LIN {X 33.675,Y 43.444,Z 52.000,A 180.000,B 0.000,C 180.000} C_DIS
LIN {X 33.433,Y 43.340,Z 52.000,A 180.000,B 0.000,C 180.000} C_DIS
LIN {X 33.269,Y 43.266,Z 52.000,A 180.000,B 0.000,C 180.000} C_DIS
LIN {X 32.897,Y 43.076,Z 52.000,A 180.000,B 0.000,C 180.000} C_DIS
LIN {X 32.718,Y 42.971,Z 52.000,A 180.000,B 0.000,C 180.000} C_DIS
LIN {X 32.539,Y 42.865,Z 52.000,A 180.000,B 0.000,C 180.000} C_DIS
LIN {X 32.361,Y 42.749,Z 52.000,A 180.000,B 0.000,C 180.000} C_DIS
LIN {X 32.182,Y 42.627,Z 52.000,A 180.000,B 0.000,C 180.000} C_DIS
LIN {X 32.072,Y 42.550,Z 52.000,A 180.000,B 0.000,C 180.000} C_DIS
LIN {X 31.824,Y 42.359,Z 52.000,A 180.000,B 0.000,C 180.000} C_DIS
LIN {X 31.646,Y 42.212,Z 52.000,A 180.000,B 0.000,C 180.000} C_DIS
LIN {X 31.421,Y 42.014,Z 52.000,A 180.000,B 0.000,C 180.000} C_DIS
LIN {X 31.288,Y 41.888,Z 52.000,A 180.000,B 0.000,C 180.000} C_DIS
LIN {X 31.057,Y 41.657,Z 52.000,A 180.000,B 0.000,C 180.000} C_DIS
LIN {X 30.930,Y 41.516,Z 52.000,A 180.000,B 0.000,C 180.000} C_DIS
LIN {X 30.739,Y 41.299,Z 52.000,A 180.000,B 0.000,C 180.000} C_DIS
LIN {X 30.598,Y 41.120,Z 52.000,A 180.000,B 0.000,C 180.000} C_DIS
LIN {X 30.460,Y 40.942,Z 52.000,A 180.000,B 0.000,C 180.000} C_DIS
LIN {X 30.394,Y 40.850,Z 52.000,A 180.000,B 0.000,C 180.000} C_DIS
LIN {X 30.213,Y 40.584,Z 52.000,A 180.000,B 0.000,C 180.000} C_DIS
LIN {X 30.102,Y 40.405,Z 52.000,A 180.000,B 0.000,C 180.000} C_DIS
LIN {X 29.996,Y 40.226,Z 52.000,A 180.000,B 0.000,C 180.000} C_DIS
LIN {X 29.896,Y 40.048,Z 52.000,A 180.000,B 0.000,C 180.000} C_DIS
LIN {X 29.805,Y 39.869,Z 52.000,A 180.000,B 0.000,C 180.000} C_DIS
LIN {X 29.714,Y 39.690,Z 52.000,A 180.000,B 0.000,C 180.000} C_DIS
LIN {X 29.559,Y 39.333,Z 52.000,A 180.000,B 0.000,C 180.000} C_DIS
LIN {X 29.500,Y 39.184,Z 52.000,A 180.000,B 0.000,C 180.000} C_DIS
LIN {X 29.425,Y 38.975,Z 52.000,A 180.000,B 0.000,C 180.000} C_DIS
LIN {X 29.362,Y 38.796,Z 52.000,A 180.000,B 0.000,C 180.000} C_DIS
LIN {X 29.258,Y 38.439,Z 52.000,A 180.000,B 0.000,C 180.000} C_DIS
LIN {X 29.213,Y 38.260,Z 52.000,A 180.000,B 0.000,C 180.000} C_DIS
LIN {X 29.143,Y 37.944,Z 52.000,A 180.000,B 0.000,C 180.000} C_DIS
LIN {X 29.134,Y 37.902,Z 52.000,A 180.000,B 0.000,C 180.000} C_DIS
LIN {X 29.077,Y 37.545,Z 52.000,A 180.000,B 0.000,C 180.000} C_DIS
LIN {X 29.053,Y 37.366,Z 52.000,A 180.000,B 0.000,C 180.000} C_DIS
LIN {X 29.020,Y 37.009,Z 52.000,A 180.000,B 0.000,C 180.000} C_DIS
LIN {X 29.012,Y 36.830,Z 52.000,A 180.000,B 0.000,C 180.000} C_DIS
LIN {X 29.006,Y 36.651,Z 52.000,A 180.000,B 0.000,C 180.000} C_DIS
LIN {X 29.002,Y 36.472,Z 52.000,A 180.000,B 0.000,C 180.000} C_DIS
LIN {X 29.013,Y 36.115,Z 52.000,A 180.000,B 0.000,C 180.000} C_DIS
LIN {X 29.025,Y 35.936,Z 52.000,A 180.000,B 0.000,C 180.000} C_DIS
LIN {X 29.059,Y 35.578,Z 52.000,A 180.000,B 0.000,C 180.000} C_DIS
LIN {X 29.086,Y 35.400,Z 52.000,A 180.000,B 0.000,C 180.000} C_DIS
LIN {X 29.114,Y 35.221,Z 52.000,A 180.000,B 0.000,C 180.000} C_DIS
LIN {X 29.143,Y 35.056,Z 52.000,A 180.000,B 0.000,C 180.000} C_DIS
LIN {X 29.226,Y 34.685,Z 52.000,A 180.000,B 0.000,C 180.000} C_DIS
LIN {X 29.274,Y 34.506,Z 52.000,A 180.000,B 0.000,C 180.000} C_DIS
LIN {X 29.326,Y 34.327,Z 52.000,A 180.000,B 0.000,C 180.000} C_DIS
LIN {X 29.381,Y 34.148,Z 52.000,A 180.000,B 0.000,C 180.000} C_DIS
LIN {X 29.509,Y 33.791,Z 52.000,A 180.000,B 0.000,C 180.000} C_DIS
LIN {X 29.583,Y 33.612,Z 52.000,A 180.000,B 0.000,C 180.000} C_DIS
LIN {X 29.679,Y 33.390,Z 52.000,A 180.000,B 0.000,C 180.000} C_DIS
LIN {X 29.742,Y 33.254,Z 52.000,A 180.000,B 0.000,C 180.000} C_DIS
LIN {X 29.924,Y 32.897,Z 52.000,A 180.000,B 0.000,C 180.000} C_DIS
LIN {X 30.029,Y 32.718,Z 52.000,A 180.000,B 0.000,C 180.000} C_DIS
LIN {X 30.135,Y 32.539,Z 52.000,A 180.000,B 0.000,C 180.000} C_DIS
LIN {X 30.215,Y 32.413,Z 52.000,A 180.000,B 0.000,C 180.000} C_DIS
LIN {X 30.394,Y 32.150,Z 52.000,A 180.000,B 0.000,C 180.000} C_DIS
LIN {X 30.503,Y 32.003,Z 52.000,A 180.000,B 0.000,C 180.000} C_DIS
LIN {X 30.641,Y 31.824,Z 52.000,A 180.000,B 0.000,C 180.000} C_DIS
LIN {X 30.752,Y 31.687,Z 52.000,A 180.000,B 0.000,C 180.000} C_DIS
LIN {X 30.945,Y 31.467,Z 52.000,A 180.000,B 0.000,C 180.000} C_DIS
LIN {X 31.109,Y 31.291,Z 52.000,A 180.000,B 0.000,C 180.000} C_DIS
LIN {X 31.291,Y 31.109,Z 52.000,A 180.000,B 0.000,C 180.000} C_DIS
LIN {X 31.467,Y 30.945,Z 52.000,A 180.000,B 0.000,C 180.000} C_DIS
LIN {X 31.687,Y 30.752,Z 52.000,A 180.000,B 0.000,C 180.000} C_DIS
LIN {X 31.824,Y 30.641,Z 52.000,A 180.000,B 0.000,C 180.000} C_DIS
LIN {X 32.003,Y 30.503,Z 52.000,A 180.000,B 0.000,C 180.000} C_DIS
LIN {X 32.150,Y 30.394,Z 52.000,A 180.000,B 0.000,C 180.000} C_DIS
LIN {X 32.413,Y 30.215,Z 52.000,A 180.000,B 0.000,C 180.000} C_DIS
LIN {X 32.539,Y 30.135,Z 52.000,A 180.000,B 0.000,C 180.000} C_DIS
LIN {X 32.718,Y 30.029,Z 52.000,A 180.000,B 0.000,C 180.000} C_DIS
LIN {X 32.897,Y 29.924,Z 52.000,A 180.000,B 0.000,C 180.000} C_DIS
LIN {X 33.254,Y 29.742,Z 52.000,A 180.000,B 0.000,C 180.000} C_DIS
LIN {X 33.390,Y 29.679,Z 52.000,A 180.000,B 0.000,C 180.000} C_DIS
LIN {X 33.612,Y 29.583,Z 52.000,A 180.000,B 0.000,C 180.000} C_DIS
LIN {X 33.791,Y 29.509,Z 52.000,A 180.000,B 0.000,C 180.000} C_DIS
LIN {X 34.148,Y 29.381,Z 52.000,A 180.000,B 0.000,C 180.000} C_DIS
LIN {X 34.327,Y 29.326,Z 52.000,A 180.000,B 0.000,C 180.000} C_DIS
LIN {X 34.506,Y 29.274,Z 52.000,A 180.000,B 0.000,C 180.000} C_DIS
LIN {X 34.685,Y 29.226,Z 52.000,A 180.000,B 0.000,C 180.000} C_DIS
LIN {X 35.056,Y 29.143,Z 52.000,A 180.000,B 0.000,C 180.000} C_DIS
LIN {X 35.221,Y 29.114,Z 52.000,A 180.000,B 0.000,C 180.000} C_DIS
LIN {X 35.400,Y 29.086,Z 52.000,A 180.000,B 0.000,C 180.000} C_DIS
LIN {X 35.578,Y 29.059,Z 52.000,A 180.000,B 0.000,C 180.000} C_DIS
LIN {X 35.936,Y 29.025,Z 52.000,A 180.000,B 0.000,C 180.000} C_DIS
LIN {X 36.115,Y 29.013,Z 52.000,A 180.000,B 0.000,C 180.000} C_DIS
LIN {X 36.472,Y 29.002,Z 52.000,A 180.000,B 0.000,C 180.000} C_DIS
LIN {X 36.651,Y 29.006,Z 52.000,A 180.000,B 0.000,C 180.000} C_DIS
LIN {X 36.830,Y 29.012,Z 52.000,A 180.000,B 0.000,C 180.000} C_DIS
LIN {X 37.009,Y 29.020,Z 52.000,A 180.000,B 0.000,C 180.000} C_DIS
LIN {X 37.366,Y 29.053,Z 52.000,A 180.000,B 0.000,C 180.000} C_DIS
LIN {X 37.545,Y 29.077,Z 52.000,A 180.000,B 0.000,C 180.000} C_DIS
LIN {X 37.902,Y 29.134,Z 52.000,A 180.000,B 0.000,C 180.000} C_DIS
LIN {X 37.944,Y 29.143,Z 52.000,A 180.000,B 0.000,C 180.000} C_DIS
LIN {X 38.260,Y 29.213,Z 52.000,A 180.000,B 0.000,C 180.000} C_DIS
LIN {X 38.439,Y 29.258,Z 52.000,A 180.000,B 0.000,C 180.000} C_DIS
LIN {X 38.796,Y 29.362,Z 52.000,A 180.000,B 0.000,C 180.000} C_DIS
LIN {X 38.975,Y 29.425,Z 52.000,A 180.000,B 0.000,C 180.000} C_DIS
LIN {X 39.184,Y 29.500,Z 52.000,A 180.000,B 0.000,C 180.000} C_DIS
LIN {X 39.333,Y 29.559,Z 52.000,A 180.000,B 0.000,C 180.000} C_DIS
LIN {X 39.690,Y 29.714,Z 52.000,A 180.000,B 0.000,C 180.000} C_DIS
LIN {X 39.869,Y 29.805,Z 52.000,A 180.000,B 0.000,C 180.000} C_DIS
LIN {X 40.048,Y 29.896,Z 52.000,A 180.000,B 0.000,C 180.000} C_DIS
LIN {X 40.226,Y 29.996,Z 52.000,A 180.000,B 0.000,C 180.000} C_DIS
LIN {X 40.405,Y 30.102,Z 52.000,A 180.000,B 0.000,C 180.000} C_DIS
LIN {X 40.584,Y 30.213,Z 52.000,A 180.000,B 0.000,C 180.000} C_DIS
LIN {X 40.850,Y 30.394,Z 52.000,A 180.000,B 0.000,C 180.000} C_DIS
LIN {X 40.942,Y 30.460,Z 52.000,A 180.000,B 0.000,C 180.000} C_DIS
LIN {X 41.120,Y 30.598,Z 52.000,A 180.000,B 0.000,C 180.000} C_DIS
LIN {X 41.299,Y 30.739,Z 52.000,A 180.000,B 0.000,C 180.000} C_DIS
LIN {X 41.516,Y 30.930,Z 52.000,A 180.000,B 0.000,C 180.000} C_DIS
LIN {X 41.657,Y 31.057,Z 52.000,A 180.000,B 0.000,C 180.000} C_DIS
LIN {X 41.888,Y 31.288,Z 52.000,A 180.000,B 0.000,C 180.000} C_DIS
LIN {X 42.014,Y 31.421,Z 52.000,A 180.000,B 0.000,C 180.000} C_DIS
LIN {X 42.212,Y 31.646,Z 52.000,A 180.000,B 0.000,C 180.000} C_DIS
LIN {X 42.359,Y 31.824,Z 52.000,A 180.000,B 0.000,C 180.000} C_DIS
LIN {X 42.550,Y 32.072,Z 52.000,A 180.000,B 0.000,C 180.000} C_DIS
LIN {X 42.627,Y 32.182,Z 52.000,A 180.000,B 0.000,C 180.000} C_DIS
LIN {X 42.749,Y 32.361,Z 52.000,A 180.000,B 0.000,C 180.000} C_DIS
LIN {X 42.865,Y 32.539,Z 52.000,A 180.000,B 0.000,C 180.000} C_DIS
LIN {X 42.971,Y 32.718,Z 52.000,A 180.000,B 0.000,C 180.000} C_DIS
LIN {X 43.076,Y 32.897,Z 52.000,A 180.000,B 0.000,C 180.000} C_DIS
LIN {X 43.266,Y 33.269,Z 52.000,A 180.000,B 0.000,C 180.000} C_DIS
LIN {X 43.340,Y 33.433,Z 52.000,A 180.000,B 0.000,C 180.000} C_DIS
LIN {X 43.444,Y 33.675,Z 52.000,A 180.000,B 0.000,C 180.000} C_DIS
LIN {X 43.491,Y 33.791,Z 52.000,A 180.000,B 0.000,C 180.000} C_DIS
LIN {X 43.623,Y 34.159,Z 52.000,A 180.000,B 0.000,C 180.000} C_DIS
LIN {X 43.674,Y 34.327,Z 52.000,A 180.000,B 0.000,C 180.000} C_DIS
LIN {X 43.726,Y 34.506,Z 52.000,A 180.000,B 0.000,C 180.000} C_DIS
LIN {X 43.774,Y 34.685,Z 52.000,A 180.000,B 0.000,C 180.000} C_DIS
LIN {X 43.854,Y 35.042,Z 52.000,A 180.000,B 0.000,C 180.000} C_DIS
LIN {X 43.886,Y 35.221,Z 52.000,A 180.000,B 0.000,C 180.000} C_DIS
LIN {X 43.914,Y 35.400,Z 52.000,A 180.000,B 0.000,C 180.000} C_DIS
LIN {X 43.941,Y 35.578,Z 52.000,A 180.000,B 0.000,C 180.000} C_DIS
LIN {X 43.981,Y 35.994,Z 52.000,A 180.000,B 0.000,C 180.000} C_DIS
LIN {X 43.987,Y 36.115,Z 52.000,A 180.000,B 0.000,C 180.000} C_DIS
LIN {X 43.998,Y 36.472,Z 52.000,A 180.000,B 0.000,C 180.000} C_DIS
LIN {X 43.994,Y 36.651,Z 52.000,A 180.000,B 0.000,C 180.000} C_DIS
LIN {X 43.988,Y 36.830,Z 52.000,A 180.000,B 0.000,C 180.000} C_DIS
LIN {X 43.981,Y 37.006,Z 52.000,A 180.000,B 0.000,C 180.000} C_DIS
LIN {X 43.947,Y 37.366,Z 52.000,A 180.000,B 0.000,C 180.000} C_DIS
LIN {X 43.923,Y 37.545,Z 52.000,A 180.000,B 0.000,C 180.000} C_DIS
LIN {X 43.866,Y 37.902,Z 52.000,A 180.000,B 0.000,C 180.000} C_DIS
LIN {X 43.827,Y 38.081,Z 52.000,A 180.000,B 0.000,C 180.000} C_DIS
LIN {X 43.787,Y 38.260,Z 52.000,A 180.000,B 0.000,C 180.000} C_DIS
LIN {X 43.742,Y 38.439,Z 52.000,A 180.000,B 0.000,C 180.000} C_DIS
LIN {X 43.638,Y 38.796,Z 52.000,A 180.000,B 0.000,C 180.000} C_DIS
LIN {X 43.623,Y 38.841,Z 52.000,A 180.000,B 0.000,C 180.000} C_DIS
LIN {X 43.511,Y 39.154,Z 52.000,A 180.000,B 0.000,C 180.000} C_DIS
LIN {X 43.444,Y 39.325,Z 52.000,A 180.000,B 0.000,C 180.000} C_DIS
LIN {X 43.286,Y 39.690,Z 52.000,A 180.000,B 0.000,C 180.000} C_DIS
LIN {X 43.266,Y 39.731,Z 52.000,A 180.000,B 0.000,C 180.000} C_DIS
LIN {X 43.087,Y 40.082,Z 52.000,A 180.000,B 0.000,C 180.000} C_DIS
LIN {X 43.004,Y 40.226,Z 52.000,A 180.000,B 0.000,C 180.000} C_DIS
LIN {X 42.898,Y 40.405,Z 52.000,A 180.000,B 0.000,C 180.000} C_DIS
LIN {X 42.787,Y 40.584,Z 52.000,A 180.000,B 0.000,C 180.000} C_DIS
LIN {X 42.665,Y 40.763,Z 52.000,A 180.000,B 0.000,C 180.000} C_DIS
LIN {X 42.550,Y 40.928,Z 52.000,A 180.000,B 0.000,C 180.000} C_DIS
LIN {X 42.372,Y 41.159,Z 52.000,A 180.000,B 0.000,C 180.000} C_DIS
LIN {X 42.261,Y 41.299,Z 52.000,A 180.000,B 0.000,C 180.000} C_DIS
LIN {X 42.014,Y 41.579,Z 52.000,A 180.000,B 0.000,C 180.000} C_DIS
LIN {X 41.943,Y 41.657,Z 52.000,A 180.000,B 0.000,C 180.000} C_DIS
LIN {X 41.657,Y 41.943,Z 52.000,A 180.000,B 0.000,C 180.000} C_DIS
LIN {X 41.579,Y 42.014,Z 52.000,A 180.000,B 0.000,C 180.000} C_DIS
LIN {X 41.323,Y 42.240,Z 52.000,A 180.000,B 0.000,C 180.000} C_DIS
; Lead Out Move Starts
LIN {X 40.878,Y 42.351,Z 52.000,A 180.000,B 0.000,C 180.000} C_DIS
LIN {X 40.529,Y 42.051,Z 52.000,A 180.000,B 0.000,C 180.000} C_DIS
LIN {X 40.187,Y 41.203,Z 52.000,A 180.000,B 0.000,C 180.000} C_DIS
LIN {X 40.055,Y 40.875,Z 52.146,A 180.000,B 0.000,C 180.000} C_DIS
LIN {X 40.000,Y 40.739,Z 52.500,A 180.000,B 0.000,C 180.000} C_DIS
; Rapid Move Starts
LIN {X 40.000,Y 40.739,Z 95.000,A 180.000,B 0.000,C 180.000} C_DIS
LIN {X 36.380,Y 112.331,Z 95.000,A 180.000,B 0.000,C 180.000} C_DIS
LIN {X 36.380,Y 112.331,Z 58.498,A 180.000,B 0.000,C 180.000} C_DIS
; Plunge Move Starts
$VEL.CP=0.01
LIN {X 36.380,Y 112.331,Z 57.625,A 180.000,B 0.000,C 180.000} C_DIS
; Lead In Move Starts
LIN {X 36.380,Y 112.331,Z 56.500,A 180.000,B 0.000,C 180.000} C_DIS
LIN {X 36.394,Y 112.185,Z 56.146,A 180.000,B 0.000,C 180.000} C_DIS
LIN {X 36.427,Y 111.833,Z 56.000,A 180.000,B 0.000,C 180.000} C_DIS
LIN {X 36.461,Y 111.470,Z 56.000,A 180.000,B 0.000,C 180.000} C_DIS
LIN {X 36.640,Y 111.132,Z 56.000,A 180.000,B 0.000,C 180.000} C_DIS
LIN {X 37.006,Y 111.019,Z 56.000,A 180.000,B 0.000,C 180.000} C_DIS
; Cutting Move Starts
$VEL.CP=0.02
LIN {X 37.366,Y 111.053,Z 56.000,A 180.000,B 0.000,C 180.000} C_DIS
LIN {X 37.545,Y 111.077,Z 56.000,A 180.000,B 0.000,C 180.000} C_DIS
LIN {X 37.902,Y 111.134,Z 56.000,A 180.000,B 0.000,C 180.000} C_DIS
LIN {X 38.081,Y 111.173,Z 56.000,A 180.000,B 0.000,C 180.000} C_DIS
LIN {X 38.260,Y 111.213,Z 56.000,A 180.000,B 0.000,C 180.000} C_DIS
LIN {X 38.439,Y 111.258,Z 56.000,A 180.000,B 0.000,C 180.000} C_DIS
LIN {X 38.796,Y 111.362,Z 56.000,A 180.000,B 0.000,C 180.000} C_DIS
LIN {X 38.841,Y 111.377,Z 56.000,A 180.000,B 0.000,C 180.000} C_DIS
LIN {X 39.154,Y 111.489,Z 56.000,A 180.000,B 0.000,C 180.000} C_DIS
LIN {X 39.325,Y 111.556,Z 56.000,A 180.000,B 0.000,C 180.000} C_DIS
LIN {X 39.690,Y 111.714,Z 56.000,A 180.000,B 0.000,C 180.000} C_DIS
LIN {X 39.731,Y 111.734,Z 56.000,A 180.000,B 0.000,C 180.000} C_DIS
LIN {X 40.082,Y 111.913,Z 56.000,A 180.000,B 0.000,C 180.000} C_DIS
LIN {X 40.226,Y 111.996,Z 56.000,A 180.000,B 0.000,C 180.000} C_DIS
LIN {X 40.405,Y 112.102,Z 56.000,A 180.000,B 0.000,C 180.000} C_DIS
LIN {X 40.584,Y 112.213,Z 56.000,A 180.000,B 0.000,C 180.000} C_DIS
LIN {X 40.763,Y 112.335,Z 56.000,A 180.000,B 0.000,C 180.000} C_DIS
LIN {X 40.928,Y 112.450,Z 56.000,A 180.000,B 0.000,C 180.000} C_DIS
LIN {X 41.159,Y 112.628,Z 56.000,A 180.000,B 0.000,C 180.000} C_DIS
LIN {X 41.299,Y 112.739,Z 56.000,A 180.000,B 0.000,C 180.000} C_DIS
LIN {X 41.579,Y 112.986,Z 56.000,A 180.000,B 0.000,C 180.000} C_DIS
LIN {X 41.657,Y 113.057,Z 56.000,A 180.000,B 0.000,C 180.000} C_DIS
LIN {X 41.943,Y 113.343,Z 56.000,A 180.000,B 0.000,C 180.000} C_DIS
LIN {X 42.014,Y 113.421,Z 56.000,A 180.000,B 0.000,C 180.000} C_DIS
LIN {X 42.261,Y 113.701,Z 56.000,A 180.000,B 0.000,C 180.000} C_DIS
LIN {X 42.372,Y 113.841,Z 56.000,A 180.000,B 0.000,C 180.000} C_DIS
LIN {X 42.550,Y 114.072,Z 56.000,A 180.000,B 0.000,C 180.000} C_DIS
LIN {X 42.665,Y 114.237,Z 56.000,A 180.000,B 0.000,C 180.000} C_DIS
LIN {X 42.787,Y 114.416,Z 56.000,A 180.000,B 0.000,C 180.000} C_DIS
LIN {X 42.898,Y 114.595,Z 56.000,A 180.000,B 0.000,C 180.000} C_DIS
LIN {X 43.004,Y 114.774,Z 56.000,A 180.000,B 0.000,C 180.000} C_DIS
LIN {X 43.087,Y 114.918,Z 56.000,A 180.000,B 0.000,C 180.000} C_DIS
LIN {X 43.266,Y 115.269,Z 56.000,A 180.000,B 0.000,C 180.000} C_DIS
LIN {X 43.286,Y 115.310,Z 56.000,A 180.000,B 0.000,C 180.000} C_DIS
LIN {X 43.444,Y 115.675,Z 56.000,A 180.000,B 0.000,C 180.000} C_DIS
LIN {X 43.511,Y 115.846,Z 56.000,A 180.000,B 0.000,C 180.000} C_DIS
LIN {X 43.623,Y 116.159,Z 56.000,A 180.000,B 0.000,C 180.000} C_DIS
LIN {X 43.638,Y 116.204,Z 56.000,A 180.000,B 0.000,C 180.000} C_DIS
LIN {X 43.742,Y 116.561,Z 56.000,A 180.000,B 0.000,C 180.000} C_DIS
LIN {X 43.787,Y 116.740,Z 56.000,A 180.000,B 0.000,C 180.000} C_DIS
LIN {X 43.827,Y 116.919,Z 56.000,A 180.000,B 0.000,C 180.000} C_DIS
LIN {X 43.866,Y 117.098,Z 56.000,A 180.000,B 0.000,C 180.000} C_DIS
LIN {X 43.923,Y 117.455,Z 56.000,A 180.000,B 0.000,C 180.000} C_DIS
LIN {X 43.947,Y 117.634,Z 56.000,A 180.000,B 0.000,C 180.000} C_DIS
LIN {X 43.981,Y 117.994,Z 56.000,A 180.000,B 0.000,C 180.000} C_DIS
LIN {X 43.988,Y 118.170,Z 56.000,A 180.000,B 0.000,C 180.000} C_DIS
LIN {X 43.994,Y 118.349,Z 56.000,A 180.000,B 0.000,C 180.000} C_DIS
LIN {X 43.998,Y 118.528,Z 56.000,A 180.000,B 0.000,C 180.000} C_DIS
LIN {X 43.987,Y 118.885,Z 56.000,A 180.000,B 0.000,C 180.000} C_DIS
LIN {X 43.981,Y 119.006,Z 56.000,A 180.000,B 0.000,C 180.000} C_DIS
LIN {X 43.941,Y 119.422,Z 56.000,A 180.000,B 0.000,C 180.000} C_DIS
LIN {X 43.914,Y 119.600,Z 56.000,A 180.000,B 0.000,C 180.000} C_DIS
LIN {X 43.886,Y 119.779,Z 56.000,A 180.000,B 0.000,C 180.000} C_DIS
LIN {X 43.854,Y 119.958,Z 56.000,A 180.000,B 0.000,C 180.000} C_DIS
LIN {X 43.774,Y 120.315,Z 56.000,A 180.000,B 0.000,C 180.000} C_DIS
LIN {X 43.726,Y 120.494,Z 56.000,A 180.000,B 0.000,C 180.000} C_DIS
LIN {X 43.674,Y 120.673,Z 56.000,A 180.000,B 0.000,C 180.000} C_DIS
LIN {X 43.623,Y 120.841,Z 56.000,A 180.000,B 0.000,C 180.000} C_DIS
LIN {X 43.491,Y 121.209,Z 56.000,A 180.000,B 0.000,C 180.000} C_DIS
LIN {X 43.444,Y 121.325,Z 56.000,A 180.000,B 0.000,C 180.000} C_DIS
LIN {X 43.340,Y 121.567,Z 56.000,A 180.000,B 0.000,C 180.000} C_DIS
LIN {X 43.266,Y 121.731,Z 56.000,A 180.000,B 0.000,C 180.000} C_DIS
LIN {X 43.076,Y 122.103,Z 56.000,A 180.000,B 0.000,C 180.000} C_DIS
LIN {X 42.971,Y 122.282,Z 56.000,A 180.000,B 0.000,C 180.000} C_DIS
LIN {X 42.865,Y 122.461,Z 56.000,A 180.000,B 0.000,C 180.000} C_DIS
LIN {X 42.749,Y 122.639,Z 56.000,A 180.000,B 0.000,C 180.000} C_DIS
LIN {X 42.627,Y 122.818,Z 56.000,A 180.000,B 0.000,C 180.000} C_DIS
LIN {X 42.550,Y 122.928,Z 56.000,A 180.000,B 0.000,C 180.000} C_DIS
LIN {X 42.359,Y 123.176,Z 56.000,A 180.000,B 0.000,C 180.000} C_DIS
LIN {X 42.212,Y 123.354,Z 56.000,A 180.000,B 0.000,C 180.000} C_DIS
LIN {X 42.014,Y 123.579,Z 56.000,A 180.000,B 0.000,C 180.000} C_DIS
LIN {X 41.888,Y 123.712,Z 56.000,A 180.000,B 0.000,C 180.000} C_DIS
LIN {X 41.657,Y 123.943,Z 56.000,A 180.000,B 0.000,C 180.000} C_DIS
LIN {X 41.516,Y 124.070,Z 56.000,A 180.000,B 0.000,C 180.000} C_DIS
LIN {X 41.299,Y 124.261,Z 56.000,A 180.000,B 0.000,C 180.000} C_DIS
LIN {X 41.120,Y 124.402,Z 56.000,A 180.000,B 0.000,C 180.000} C_DIS
LIN {X 40.942,Y 124.540,Z 56.000,A 180.000,B 0.000,C 180.000} C_DIS
LIN {X 40.850,Y 124.606,Z 56.000,A 180.000,B 0.000,C 180.000} C_DIS
LIN {X 40.584,Y 124.787,Z 56.000,A 180.000,B 0.000,C 180.000} C_DIS
LIN {X 40.405,Y 124.898,Z 56.000,A 180.000,B 0.000,C 180.000} C_DIS
LIN {X 40.226,Y 125.004,Z 56.000,A 180.000,B 0.000,C 180.000} C_DIS
LIN {X 40.048,Y 125.104,Z 56.000,A 180.000,B 0.000,C 180.000} C_DIS
LIN {X 39.869,Y 125.195,Z 56.000,A 180.000,B 0.000,C 180.000} C_DIS
LIN {X 39.690,Y 125.286,Z 56.000,A 180.000,B 0.000,C 180.000} C_DIS
LIN {X 39.333,Y 125.441,Z 56.000,A 180.000,B 0.000,C 180.000} C_DIS
LIN {X 39.184,Y 125.500,Z 56.000,A 180.000,B 0.000,C 180.000} C_DIS
LIN {X 38.975,Y 125.575,Z 56.000,A 180.000,B 0.000,C 180.000} C_DIS
LIN {X 38.796,Y 125.638,Z 56.000,A 180.000,B 0.000,C 180.000} C_DIS
LIN {X 38.439,Y 125.742,Z 56.000,A 180.000,B 0.000,C 180.000} C_DIS
LIN {X 38.260,Y 125.787,Z 56.000,A 180.000,B 0.000,C 180.000} C_DIS
LIN {X 37.944,Y 125.857,Z 56.000,A 180.000,B 0.000,C 180.000} C_DIS
LIN {X 37.902,Y 125.866,Z 56.000,A 180.000,B 0.000,C 180.000} C_DIS
LIN {X 37.545,Y 125.923,Z 56.000,A 180.000,B 0.000,C 180.000} C_DIS
LIN {X 37.366,Y 125.947,Z 56.000,A 180.000,B 0.000,C 180.000} C_DIS
LIN {X 37.009,Y 125.980,Z 56.000,A 180.000,B 0.000,C 180.000} C_DIS
LIN {X 36.830,Y 125.988,Z 56.000,A 180.000,B 0.000,C 180.000} C_DIS
LIN {X 36.651,Y 125.994,Z 56.000,A 180.000,B 0.000,C 180.000} C_DIS
LIN {X 36.472,Y 125.998,Z 56.000,A 180.000,B 0.000,C 180.000} C_DIS
LIN {X 36.115,Y 125.987,Z 56.000,A 180.000,B 0.000,C 180.000} C_DIS
LIN {X 35.936,Y 125.975,Z 56.000,A 180.000,B 0.000,C 180.000} C_DIS
LIN {X 35.578,Y 125.941,Z 56.000,A 180.000,B 0.000,C 180.000} C_DIS
LIN {X 35.400,Y 125.914,Z 56.000,A 180.000,B 0.000,C 180.000} C_DIS
LIN {X 35.221,Y 125.886,Z 56.000,A 180.000,B 0.000,C 180.000} C_DIS
LIN {X 35.056,Y 125.857,Z 56.000,A 180.000,B 0.000,C 180.000} C_DIS
LIN {X 34.685,Y 125.774,Z 56.000,A 180.000,B 0.000,C 180.000} C_DIS
LIN {X 34.506,Y 125.726,Z 56.000,A 180.000,B 0.000,C 180.000} C_DIS
LIN {X 34.327,Y 125.674,Z 56.000,A 180.000,B 0.000,C 180.000} C_DIS
LIN {X 34.148,Y 125.619,Z 56.000,A 180.000,B 0.000,C 180.000} C_DIS
LIN {X 33.791,Y 125.491,Z 56.000,A 180.000,B 0.000,C 180.000} C_DIS
LIN {X 33.612,Y 125.417,Z 56.000,A 180.000,B 0.000,C 180.000} C_DIS
LIN {X 33.390,Y 125.321,Z 56.000,A 180.000,B 0.000,C 180.000} C_DIS
LIN {X 33.254,Y 125.258,Z 56.000,A 180.000,B 0.000,C 180.000} C_DIS
LIN {X 32.897,Y 125.076,Z 56.000,A 180.000,B 0.000,C 180.000} C_DIS
LIN {X 32.718,Y 124.971,Z 56.000,A 180.000,B 0.000,C 180.000} C_DIS
LIN {X 32.539,Y 124.865,Z 56.000,A 180.000,B 0.000,C 180.000} C_DIS
LIN {X 32.413,Y 124.785,Z 56.000,A 180.000,B 0.000,C 180.000} C_DIS
LIN {X 32.150,Y 124.606,Z 56.000,A 180.000,B 0.000,C 180.000} C_DIS
LIN {X 32.003,Y 124.497,Z 56.000,A 180.000,B 0.000,C 180.000} C_DIS
LIN {X 31.824,Y 124.359,Z 56.000,A 180.000,B 0.000,C 180.000} C_DIS
LIN {X 31.687,Y 124.248,Z 56.000,A 180.000,B 0.000,C 180.000} C_DIS
LIN {X 31.467,Y 124.055,Z 56.000,A 180.000,B 0.000,C 180.000} C_DIS
LIN {X 31.291,Y 123.891,Z 56.000,A 180.000,B 0.000,C 180.000} C_DIS
LIN {X 31.109,Y 123.709,Z 56.000,A 180.000,B 0.000,C 180.000} C_DIS
LIN {X 30.945,Y 123.533,Z 56.000,A 180.000,B 0.000,C 180.000} C_DIS
LIN {X 30.752,Y 123.313,Z 56.000,A 180.000,B 0.000,C 180.000} C_DIS
LIN {X 30.641,Y 123.176,Z 56.000,A 180.000,B 0.000,C 180.000} C_DIS
LIN {X 30.503,Y 122.997,Z 56.000,A 180.000,B 0.000,C 180.000} C_DIS
LIN {X 30.394,Y 122.850,Z 56.000,A 180.000,B 0.000,C 180.000} C_DIS
LIN {X 30.215,Y 122.587,Z 56.000,A 180.000,B 0.000,C 180.000} C_DIS
LIN {X 30.135,Y 122.461,Z 56.000,A 180.000,B 0.000,C 180.000} C_DIS
LIN {X 30.029,Y 122.282,Z 56.000,A 180.000,B 0.000,C 180.000} C_DIS
LIN {X 29.924,Y 122.103,Z 56.000,A 180.000,B 0.000,C 180.000} C_DIS
LIN {X 29.742,Y 121.746,Z 56.000,A 180.000,B 0.000,C 180.000} C_DIS
LIN {X 29.679,Y 121.610,Z 56.000,A 180.000,B 0.000,C 180.000} C_DIS
LIN {X 29.583,Y 121.388,Z 56.000,A 180.000,B 0.000,C 180.000} C_DIS
LIN {X 29.509,Y 121.209,Z 56.000,A 180.000,B 0.000,C 180.000} C_DIS
LIN {X 29.381,Y 120.852,Z 56.000,A 180.000,B 0.000,C 180.000} C_DIS
LIN {X 29.326,Y 120.673,Z 56.000,A 180.000,B 0.000,C 180.000} C_DIS
LIN {X 29.274,Y 120.494,Z 56.000,A 180.000,B 0.000,C 180.000} C_DIS
LIN {X 29.226,Y 120.315,Z 56.000,A 180.000,B 0.000,C 180.000} C_DIS
LIN {X 29.143,Y 119.944,Z 56.000,A 180.000,B 0.000,C 180.000} C_DIS
LIN {X 29.114,Y 119.779,Z 56.000,A 180.000,B 0.000,C 180.000} C_DIS
LIN {X 29.086,Y 119.600,Z 56.000,A 180.000,B 0.000,C 180.000} C_DIS
LIN {X 29.059,Y 119.422,Z 56.000,A 180.000,B 0.000,C 180.000} C_DIS
LIN {X 29.025,Y 119.064,Z 56.000,A 180.000,B 0.000,C 180.000} C_DIS
LIN {X 29.013,Y 118.885,Z 56.000,A 180.000,B 0.000,C 180.000} C_DIS
LIN {X 29.002,Y 118.528,Z 56.000,A 180.000,B 0.000,C 180.000} C_DIS
LIN {X 29.006,Y 118.349,Z 56.000,A 180.000,B 0.000,C 180.000} C_DIS
LIN {X 29.012,Y 118.170,Z 56.000,A 180.000,B 0.000,C 180.000} C_DIS
LIN {X 29.020,Y 117.991,Z 56.000,A 180.000,B 0.000,C 180.000} C_DIS
LIN {X 29.053,Y 117.634,Z 56.000,A 180.000,B 0.000,C 180.000} C_DIS
LIN {X 29.077,Y 117.455,Z 56.000,A 180.000,B 0.000,C 180.000} C_DIS
LIN {X 29.134,Y 117.098,Z 56.000,A 180.000,B 0.000,C 180.000} C_DIS
LIN {X 29.143,Y 117.056,Z 56.000,A 180.000,B 0.000,C 180.000} C_DIS
LIN {X 29.213,Y 116.740,Z 56.000,A 180.000,B 0.000,C 180.000} C_DIS
LIN {X 29.258,Y 116.561,Z 56.000,A 180.000,B 0.000,C 180.000} C_DIS
LIN {X 29.362,Y 116.204,Z 56.000,A 180.000,B 0.000,C 180.000} C_DIS
LIN {X 29.425,Y 116.025,Z 56.000,A 180.000,B 0.000,C 180.000} C_DIS
LIN {X 29.500,Y 115.816,Z 56.000,A 180.000,B 0.000,C 180.000} C_DIS
LIN {X 29.559,Y 115.667,Z 56.000,A 180.000,B 0.000,C 180.000} C_DIS
LIN {X 29.714,Y 115.310,Z 56.000,A 180.000,B 0.000,C 180.000} C_DIS
LIN {X 29.805,Y 115.131,Z 56.000,A 180.000,B 0.000,C 180.000} C_DIS
LIN {X 29.896,Y 114.952,Z 56.000,A 180.000,B 0.000,C 180.000} C_DIS
LIN {X 29.996,Y 114.774,Z 56.000,A 180.000,B 0.000,C 180.000} C_DIS
LIN {X 30.102,Y 114.595,Z 56.000,A 180.000,B 0.000,C 180.000} C_DIS
LIN {X 30.213,Y 114.416,Z 56.000,A 180.000,B 0.000,C 180.000} C_DIS
LIN {X 30.394,Y 114.150,Z 56.000,A 180.000,B 0.000,C 180.000} C_DIS
LIN {X 30.460,Y 114.058,Z 56.000,A 180.000,B 0.000,C 180.000} C_DIS
LIN {X 30.598,Y 113.880,Z 56.000,A 180.000,B 0.000,C 180.000} C_DIS
LIN {X 30.739,Y 113.701,Z 56.000,A 180.000,B 0.000,C 180.000} C_DIS
LIN {X 30.930,Y 113.484,Z 56.000,A 180.000,B 0.000,C 180.000} C_DIS
LIN {X 31.057,Y 113.343,Z 56.000,A 180.000,B 0.000,C 180.000} C_DIS
LIN {X 31.288,Y 113.112,Z 56.000,A 180.000,B 0.000,C 180.000} C_DIS
LIN {X 31.421,Y 112.986,Z 56.000,A 180.000,B 0.000,C 180.000} C_DIS
LIN {X 31.646,Y 112.788,Z 56.000,A 180.000,B 0.000,C 180.000} C_DIS
LIN {X 31.824,Y 112.641,Z 56.000,A 180.000,B 0.000,C 180.000} C_DIS
LIN {X 32.072,Y 112.450,Z 56.000,A 180.000,B 0.000,C 180.000} C_DIS
LIN {X 32.182,Y 112.373,Z 56.000,A 180.000,B 0.000,C 180.000} C_DIS
LIN {X 32.361,Y 112.251,Z 56.000,A 180.000,B 0.000,C 180.000} C_DIS
LIN {X 32.539,Y 112.135,Z 56.000,A 180.000,B 0.000,C 180.000} C_DIS
LIN {X 32.718,Y 112.029,Z 56.000,A 180.000,B 0.000,C 180.000} C_DIS
LIN {X 32.897,Y 111.924,Z 56.000,A 180.000,B 0.000,C 180.000} C_DIS
LIN {X 33.269,Y 111.734,Z 56.000,A 180.000,B 0.000,C 180.000} C_DIS
LIN {X 33.433,Y 111.660,Z 56.000,A 180.000,B 0.000,C 180.000} C_DIS
LIN {X 33.675,Y 111.556,Z 56.000,A 180.000,B 0.000,C 180.000} C_DIS
LIN {X 33.791,Y 111.509,Z 56.000,A 180.000,B 0.000,C 180.000} C_DIS
LIN {X 34.159,Y 111.377,Z 56.000,A 180.000,B 0.000,C 180.000} C_DIS
LIN {X 34.327,Y 111.326,Z 56.000,A 180.000,B 0.000,C 180.000} C_DIS
LIN {X 34.506,Y 111.274,Z 56.000,A 180.000,B 0.000,C 180.000} C_DIS
LIN {X 34.685,Y 111.226,Z 56.000,A 180.000,B 0.000,C 180.000} C_DIS
LIN {X 35.042,Y 111.146,Z 56.000,A 180.000,B 0.000,C 180.000} C_DIS
LIN {X 35.221,Y 111.114,Z 56.000,A 180.000,B 0.000,C 180.000} C_DIS
LIN {X 35.400,Y 111.086,Z 56.000,A 180.000,B 0.000,C 180.000} C_DIS
LIN {X 35.578,Y 111.059,Z 56.000,A 180.000,B 0.000,C 180.000} C_DIS
LIN {X 35.994,Y 111.019,Z 56.000,A 180.000,B 0.000,C 180.000} C_DIS
LIN {X 36.115,Y 111.013,Z 56.000,A 180.000,B 0.000,C 180.000} C_DIS
LIN {X 36.472,Y 111.002,Z 56.000,A 180.000,B 0.000,C 180.000} C_DIS
LIN {X 36.651,Y 111.006,Z 56.000,A 180.000,B 0.000,C 180.000} C_DIS
LIN {X 36.830,Y 111.012,Z 56.000,A 180.000,B 0.000,C 180.000} C_DIS
LIN {X 37.006,Y 111.019,Z 56.000,A 180.000,B 0.000,C 180.000} C_DIS
; Link Move Starts
LIN {X 37.320,Y 111.049,Z 56.000,A 180.000,B 0.000,C 180.000} C_DIS
LIN {X 37.632,Y 111.091,Z 55.999,A 180.000,B 0.000,C 180.000} C_DIS
LIN {X 37.943,Y 111.142,Z 55.998,A 180.000,B 0.000,C 180.000} C_DIS
LIN {X 38.250,Y 111.211,Z 55.996,A 180.000,B 0.000,C 180.000} C_DIS
LIN {X 38.554,Y 111.292,Z 55.994,A 180.000,B 0.000,C 180.000} C_DIS
LIN {X 38.856,Y 111.382,Z 55.991,A 180.000,B 0.000,C 180.000} C_DIS
LIN {X 39.152,Y 111.489,Z 55.988,A 180.000,B 0.000,C 180.000} C_DIS
LIN {X 39.444,Y 111.607,Z 55.985,A 180.000,B 0.000,C 180.000} C_DIS
LIN {X 39.732,Y 111.735,Z 55.981,A 180.000,B 0.000,C 180.000} C_DIS
LIN {X 40.013,Y 111.878,Z 55.977,A 180.000,B 0.000,C 180.000} C_DIS
LIN {X 40.287,Y 112.032,Z 55.972,A 180.000,B 0.000,C 180.000} C_DIS
LIN {X 40.423,Y 112.112,Z 55.969,A 180.000,B 0.000,C 180.000} C_DIS
LIN {X 40.557,Y 112.195,Z 55.967,A 180.000,B 0.000,C 180.000} C_DIS
LIN {X 40.687,Y 112.284,Z 55.964,A 180.000,B 0.000,C 180.000} C_DIS
LIN {X 40.818,Y 112.372,Z 55.961,A 180.000,B 0.000,C 180.000} C_DIS
LIN {X 40.946,Y 112.463,Z 55.959,A 180.000,B 0.000,C 180.000} C_DIS
LIN {X 41.071,Y 112.560,Z 55.956,A 180.000,B 0.000,C 180.000} C_DIS
LIN {X 41.195,Y 112.656,Z 55.952,A 180.000,B 0.000,C 180.000} C_DIS
LIN {X 41.317,Y 112.755,Z 55.949,A 180.000,B 0.000,C 180.000} C_DIS
LIN {X 41.436,Y 112.859,Z 55.946,A 180.000,B 0.000,C 180.000} C_DIS
LIN {X 41.554,Y 112.964,Z 55.943,A 180.000,B 0.000,C 180.000} C_DIS
LIN {X 41.670,Y 113.070,Z 55.939,A 180.000,B 0.000,C 180.000} C_DIS
LIN {X 41.781,Y 113.181,Z 55.936,A 180.000,B 0.000,C 180.000} C_DIS
LIN {X 41.892,Y 113.293,Z 55.932,A 180.000,B 0.000,C 180.000} C_DIS
LIN {X 42.001,Y 113.407,Z 55.928,A 180.000,B 0.000,C 180.000} C_DIS
LIN {X 42.106,Y 113.525,Z 55.925,A 180.000,B 0.000,C 180.000} C_DIS
LIN {X 42.210,Y 113.643,Z 55.921,A 180.000,B 0.000,C 180.000} C_DIS
LIN {X 42.311,Y 113.763,Z 55.917,A 180.000,B 0.000,C 180.000} C_DIS
LIN {X 42.408,Y 113.888,Z 55.913,A 180.000,B 0.000,C 180.000} C_DIS
LIN {X 42.504,Y 114.012,Z 55.909,A 180.000,B 0.000,C 180.000} C_DIS
LIN {X 42.598,Y 114.139,Z 55.905,A 180.000,B 0.000,C 180.000} C_DIS
LIN {X 42.687,Y 114.269,Z 55.900,A 180.000,B 0.000,C 180.000} C_DIS
LIN {X 42.775,Y 114.399,Z 55.896,A 180.000,B 0.000,C 180.000} C_DIS
LIN {X 42.861,Y 114.531,Z 55.892,A 180.000,B 0.000,C 180.000} C_DIS
LIN {X 42.941,Y 114.667,Z 55.887,A 180.000,B 0.000,C 180.000} C_DIS
LIN {X 43.021,Y 114.803,Z 55.883,A 180.000,B 0.000,C 180.000} C_DIS
LIN {X 43.098,Y 114.940,Z 55.878,A 180.000,B 0.000,C 180.000} C_DIS
LIN {X 43.169,Y 115.080,Z 55.873,A 180.000,B 0.000,C 180.000} C_DIS
LIN {X 43.241,Y 115.221,Z 55.869,A 180.000,B 0.000,C 180.000} C_DIS
LIN {X 43.309,Y 115.363,Z 55.864,A 180.000,B 0.000,C 180.000} C_DIS
LIN {X 43.372,Y 115.507,Z 55.859,A 180.000,B 0.000,C 180.000} C_DIS
LIN {X 43.434,Y 115.652,Z 55.854,A 180.000,B 0.000,C 180.000} C_DIS
LIN {X 43.465,Y 115.724,Z 55.851,A 180.000,B 0.000,C 180.000} C_DIS
LIN {X 43.493,Y 115.798,Z 55.849,A 180.000,B 0.000,C 180.000} C_DIS
LIN {X 43.520,Y 115.872,Z 55.846,A 180.000,B 0.000,C 180.000} C_DIS
LIN {X 43.546,Y 115.946,Z 55.844,A 180.000,B 0.000,C 180.000} C_DIS
LIN {X 43.573,Y 116.020,Z 55.841,A 180.000,B 0.000,C 180.000} C_DIS
LIN {X 43.627,Y 116.168,Z 55.836,A 180.000,B 0.000,C 180.000} C_DIS
LIN {X 43.649,Y 116.244,Z 55.833,A 180.000,B 0.000,C 180.000} C_DIS
LIN {X 43.693,Y 116.395,Z 55.828,A 180.000,B 0.000,C 180.000} C_DIS
LIN {X 43.737,Y 116.546,Z 55.823,A 180.000,B 0.000,C 180.000} C_DIS
LIN {X 43.759,Y 116.622,Z 55.820,A 180.000,B 0.000,C 180.000} C_DIS
LIN {X 43.777,Y 116.698,Z 55.817,A 180.000,B 0.000,C 180.000} C_DIS
LIN {X 43.812,Y 116.852,Z 55.812,A 180.000,B 0.000,C 180.000} C_DIS
LIN {X 43.863,Y 117.083,Z 55.804,A 180.000,B 0.000,C 180.000} C_DIS
LIN {X 43.876,Y 117.160,Z 55.801,A 180.000,B 0.000,C 180.000} C_DIS
LIN {X 43.913,Y 117.394,Z 55.793,A 180.000,B 0.000,C 180.000} C_DIS
LIN {X 43.938,Y 117.549,Z 55.787,A 180.000,B 0.000,C 180.000} C_DIS
LIN {X 43.946,Y 117.628,Z 55.785,A 180.000,B 0.000,C 180.000} C_DIS
LIN {X 43.961,Y 117.784,Z 55.779,A 180.000,B 0.000,C 180.000} C_DIS
LIN {X 43.983,Y 118.020,Z 55.771,A 180.000,B 0.000,C 180.000} C_DIS
LIN {X 43.986,Y 118.098,Z 55.768,A 180.000,B 0.000,C 180.000} C_DIS
LIN {X 43.994,Y 118.334,Z 55.760,A 180.000,B 0.000,C 180.000} C_DIS
LIN {X 43.999,Y 118.492,Z 55.754,A 180.000,B 0.000,C 180.000} C_DIS
LIN {X 43.997,Y 118.571,Z 55.752,A 180.000,B 0.000,C 180.000} C_DIS
LIN {X 43.992,Y 118.728,Z 55.746,A 180.000,B 0.000,C 180.000} C_DIS
LIN {X 43.984,Y 118.964,Z 55.738,A 180.000,B 0.000,C 180.000} C_DIS
LIN {X 43.977,Y 119.043,Z 55.735,A 180.000,B 0.000,C 180.000} C_DIS
LIN {X 43.955,Y 119.278,Z 55.727,A 180.000,B 0.000,C 180.000} C_DIS
LIN {X 43.940,Y 119.435,Z 55.721,A 180.000,B 0.000,C 180.000} C_DIS
LIN {X 43.928,Y 119.513,Z 55.719,A 180.000,B 0.000,C 180.000} C_DIS
LIN {X 43.903,Y 119.668,Z 55.713,A 180.000,B 0.000,C 180.000} C_DIS
LIN {X 43.867,Y 119.901,Z 55.705,A 180.000,B 0.000,C 180.000} C_DIS
LIN {X 43.850,Y 119.978,Z 55.702,A 180.000,B 0.000,C 180.000} C_DIS
LIN {X 43.764,Y 120.363,Z 55.688,A 180.000,B 0.000,C 180.000} C_DIS
LIN {X 43.742,Y 120.438,Z 55.686,A 180.000,B 0.000,C 180.000} C_DIS
LIN {X 43.698,Y 120.590,Z 55.680,A 180.000,B 0.000,C 180.000} C_DIS
LIN {X 43.632,Y 120.817,Z 55.672,A 180.000,B 0.000,C 180.000} C_DIS
LIN {X 43.605,Y 120.891,Z 55.669,A 180.000,B 0.000,C 180.000} C_DIS
LIN {X 43.499,Y 121.187,Z 55.658,A 180.000,B 0.000,C 180.000} C_DIS
LIN {X 43.472,Y 121.261,Z 55.655,A 180.000,B 0.000,C 180.000} C_DIS
LIN {X 43.409,Y 121.406,Z 55.650,A 180.000,B 0.000,C 180.000} C_DIS
LIN {X 43.316,Y 121.623,Z 55.642,A 180.000,B 0.000,C 180.000} C_DIS
LIN {X 43.284,Y 121.695,Z 55.639,A 180.000,B 0.000,C 180.000} C_DIS
LIN {X 43.105,Y 122.046,Z 55.625,A 180.000,B 0.000,C 180.000} C_DIS
LIN {X 43.069,Y 122.116,Z 55.622,A 180.000,B 0.000,C 180.000} C_DIS
LIN {X 42.949,Y 122.319,Z 55.614,A 180.000,B 0.000,C 180.000} C_DIS
LIN {X 42.869,Y 122.455,Z 55.609,A 180.000,B 0.000,C 180.000} C_DIS
LIN {X 42.829,Y 122.522,Z 55.606,A 180.000,B 0.000,C 180.000} C_DIS
LIN {X 42.607,Y 122.848,Z 55.592,A 180.000,B 0.000,C 180.000} C_DIS
LIN {X 42.563,Y 122.913,Z 55.589,A 180.000,B 0.000,C 180.000} C_DIS
LIN {X 42.321,Y 123.224,Z 55.576,A 180.000,B 0.000,C 180.000} C_DIS
LIN {X 42.273,Y 123.286,Z 55.573,A 180.000,B 0.000,C 180.000} C_DIS
LIN {X 42.012,Y 123.581,Z 55.559,A 180.000,B 0.000,C 180.000} C_DIS
LIN {X 41.960,Y 123.640,Z 55.556,A 180.000,B 0.000,C 180.000} C_DIS
LIN {X 41.681,Y 123.918,Z 55.543,A 180.000,B 0.000,C 180.000} C_DIS
LIN {X 41.625,Y 123.974,Z 55.540,A 180.000,B 0.000,C 180.000} C_DIS
LIN {X 41.330,Y 124.234,Z 55.526,A 180.000,B 0.000,C 180.000} C_DIS
LIN {X 41.270,Y 124.286,Z 55.523,A 180.000,B 0.000,C 180.000} C_DIS
LIN {X 40.959,Y 124.527,Z 55.510,A 180.000,B 0.000,C 180.000} C_DIS
LIN {X 40.896,Y 124.575,Z 55.507,A 180.000,B 0.000,C 180.000} C_DIS
LIN {X 40.570,Y 124.796,Z 55.493,A 180.000,B 0.000,C 180.000} C_DIS
LIN {X 40.505,Y 124.839,Z 55.490,A 180.000,B 0.000,C 180.000} C_DIS
LIN {X 40.166,Y 125.040,Z 55.477,A 180.000,B 0.000,C 180.000} C_DIS
LIN {X 40.097,Y 125.079,Z 55.474,A 180.000,B 0.000,C 180.000} C_DIS
LIN {X 39.747,Y 125.258,Z 55.460,A 180.000,B 0.000,C 180.000} C_DIS
LIN {X 39.676,Y 125.292,Z 55.457,A 180.000,B 0.000,C 180.000} C_DIS
LIN {X 39.315,Y 125.449,Z 55.444,A 180.000,B 0.000,C 180.000} C_DIS
LIN {X 39.242,Y 125.479,Z 55.441,A 180.000,B 0.000,C 180.000} C_DIS
LIN {X 38.871,Y 125.612,Z 55.427,A 180.000,B 0.000,C 180.000} C_DIS
LIN {X 38.797,Y 125.638,Z 55.424,A 180.000,B 0.000,C 180.000} C_DIS
LIN {X 38.570,Y 125.704,Z 55.416,A 180.000,B 0.000,C 180.000} C_DIS
LIN {X 38.419,Y 125.748,Z 55.411,A 180.000,B 0.000,C 180.000} C_DIS
LIN {X 38.343,Y 125.768,Z 55.408,A 180.000,B 0.000,C 180.000} C_DIS
LIN {X 37.958,Y 125.854,Z 55.394,A 180.000,B 0.000,C 180.000} C_DIS
LIN {X 37.881,Y 125.870,Z 55.391,A 180.000,B 0.000,C 180.000} C_DIS
LIN {X 37.726,Y 125.894,Z 55.386,A 180.000,B 0.000,C 180.000} C_DIS
LIN {X 37.492,Y 125.931,Z 55.378,A 180.000,B 0.000,C 180.000} C_DIS
LIN {X 37.414,Y 125.942,Z 55.375,A 180.000,B 0.000,C 180.000} C_DIS
LIN {X 37.022,Y 125.979,Z 55.361,A 180.000,B 0.000,C 180.000} C_DIS
LIN {X 36.944,Y 125.985,Z 55.358,A 180.000,B 0.000,C 180.000} C_DIS
LIN {X 36.786,Y 125.990,Z 55.353,A 180.000,B 0.000,C 180.000} C_DIS
LIN {X 36.550,Y 125.997,Z 55.345,A 180.000,B 0.000,C 180.000} C_DIS
LIN {X 36.471,Y 125.998,Z 55.342,A 180.000,B 0.000,C 180.000} C_DIS
LIN {X 36.078,Y 125.985,Z 55.328,A 180.000,B 0.000,C 180.000} C_DIS
LIN {X 35.999,Y 125.981,Z 55.325,A 180.000,B 0.000,C 180.000} C_DIS
LIN {X 35.921,Y 125.974,Z 55.323,A 180.000,B 0.000,C 180.000} C_DIS
LIN {X 35.764,Y 125.959,Z 55.317,A 180.000,B 0.000,C 180.000} C_DIS
LIN {X 35.607,Y 125.944,Z 55.312,A 180.000,B 0.000,C 180.000} C_DIS
LIN {X 35.529,Y 125.935,Z 55.309,A 180.000,B 0.000,C 180.000} C_DIS
LIN {X 35.373,Y 125.910,Z 55.303,A 180.000,B 0.000,C 180.000} C_DIS
LIN {X 35.295,Y 125.898,Z 55.301,A 180.000,B 0.000,C 180.000} C_DIS
LIN {X 35.140,Y 125.873,Z 55.295,A 180.000,B 0.000,C 180.000} C_DIS
LIN {X 35.062,Y 125.859,Z 55.292,A 180.000,B 0.000,C 180.000} C_DIS
LIN {X 34.986,Y 125.842,Z 55.290,A 180.000,B 0.000,C 180.000} C_DIS
LIN {X 34.832,Y 125.807,Z 55.284,A 180.000,B 0.000,C 180.000} C_DIS
LIN {X 34.678,Y 125.773,Z 55.279,A 180.000,B 0.000,C 180.000} C_DIS
LIN {X 34.602,Y 125.754,Z 55.276,A 180.000,B 0.000,C 180.000} C_DIS
LIN {X 34.451,Y 125.710,Z 55.270,A 180.000,B 0.000,C 180.000} C_DIS
LIN {X 34.375,Y 125.688,Z 55.268,A 180.000,B 0.000,C 180.000} C_DIS
LIN {X 34.224,Y 125.644,Z 55.262,A 180.000,B 0.000,C 180.000} C_DIS
LIN {X 34.149,Y 125.620,Z 55.259,A 180.000,B 0.000,C 180.000} C_DIS
LIN {X 34.075,Y 125.593,Z 55.257,A 180.000,B 0.000,C 180.000} C_DIS
LIN {X 33.926,Y 125.539,Z 55.251,A 180.000,B 0.000,C 180.000} C_DIS
LIN {X 33.778,Y 125.486,Z 55.246,A 180.000,B 0.000,C 180.000} C_DIS
LIN {X 33.705,Y 125.457,Z 55.243,A 180.000,B 0.000,C 180.000} C_DIS
LIN {X 33.560,Y 125.395,Z 55.237,A 180.000,B 0.000,C 180.000} C_DIS
LIN {X 33.488,Y 125.363,Z 55.235,A 180.000,B 0.000,C 180.000} C_DIS
LIN {X 33.344,Y 125.301,Z 55.229,A 180.000,B 0.000,C 180.000} C_DIS
LIN {X 33.272,Y 125.267,Z 55.226,A 180.000,B 0.000,C 180.000} C_DIS
LIN {X 33.202,Y 125.232,Z 55.224,A 180.000,B 0.000,C 180.000} C_DIS
LIN {X 33.062,Y 125.160,Z 55.218,A 180.000,B 0.000,C 180.000} C_DIS
LIN {X 32.921,Y 125.089,Z 55.213,A 180.000,B 0.000,C 180.000} C_DIS
LIN {X 32.853,Y 125.051,Z 55.210,A 180.000,B 0.000,C 180.000} C_DIS
LIN {X 32.717,Y 124.970,Z 55.204,A 180.000,B 0.000,C 180.000} C_DIS
LIN {X 32.649,Y 124.930,Z 55.202,A 180.000,B 0.000,C 180.000} C_DIS
LIN {X 32.514,Y 124.850,Z 55.196,A 180.000,B 0.000,C 180.000} C_DIS
LIN {X 32.447,Y 124.808,Z 55.193,A 180.000,B 0.000,C 180.000} C_DIS
LIN {X 32.187,Y 124.631,Z 55.182,A 180.000,B 0.000,C 180.000} C_DIS
LIN {X 32.122,Y 124.586,Z 55.180,A 180.000,B 0.000,C 180.000} C_DIS
LIN {X 32.058,Y 124.540,Z 55.177,A 180.000,B 0.000,C 180.000} C_DIS
LIN {X 31.933,Y 124.443,Z 55.172,A 180.000,B 0.000,C 180.000} C_DIS
LIN {X 31.809,Y 124.347,Z 55.166,A 180.000,B 0.000,C 180.000} C_DIS
LIN {X 31.747,Y 124.299,Z 55.164,A 180.000,B 0.000,C 180.000} C_DIS
LIN {X 31.686,Y 124.248,Z 55.161,A 180.000,B 0.000,C 180.000} C_DIS
LIN {X 31.627,Y 124.196,Z 55.159,A 180.000,B 0.000,C 180.000} C_DIS
LIN {X 31.568,Y 124.144,Z 55.156,A 180.000,B 0.000,C 180.000} C_DIS
LIN {X 31.509,Y 124.092,Z 55.154,A 180.000,B 0.000,C 180.000} C_DIS
LIN {X 31.450,Y 124.040,Z 55.151,A 180.000,B 0.000,C 180.000} C_DIS
LIN {X 31.391,Y 123.988,Z 55.149,A 180.000,B 0.000,C 180.000} C_DIS
LIN {X 31.278,Y 123.878,Z 55.144,A 180.000,B 0.000,C 180.000} C_DIS
LIN {X 31.167,Y 123.766,Z 55.139,A 180.000,B 0.000,C 180.000} C_DIS
LIN {X 31.055,Y 123.655,Z 55.134,A 180.000,B 0.000,C 180.000} C_DIS
LIN {X 30.950,Y 123.538,Z 55.129,A 180.000,B 0.000,C 180.000} C_DIS
LIN {X 30.846,Y 123.420,Z 55.124,A 180.000,B 0.000,C 180.000} C_DIS
LIN {X 30.741,Y 123.302,Z 55.120,A 180.000,B 0.000,C 180.000} C_DIS
LIN {X 30.643,Y 123.179,Z 55.115,A 180.000,B 0.000,C 180.000} C_DIS
LIN {X 30.547,Y 123.054,Z 55.111,A 180.000,B 0.000,C 180.000} C_DIS
LIN {X 30.450,Y 122.930,Z 55.106,A 180.000,B 0.000,C 180.000} C_DIS
LIN {X 30.360,Y 122.800,Z 55.102,A 180.000,B 0.000,C 180.000} C_DIS
LIN {X 30.272,Y 122.670,Z 55.097,A 180.000,B 0.000,C 180.000} C_DIS
LIN {X 30.183,Y 122.540,Z 55.093,A 180.000,B 0.000,C 180.000} C_DIS
LIN {X 30.102,Y 122.405,Z 55.089,A 180.000,B 0.000,C 180.000} C_DIS
LIN {X 30.022,Y 122.269,Z 55.085,A 180.000,B 0.000,C 180.000} C_DIS
LIN {X 29.941,Y 122.134,Z 55.081,A 180.000,B 0.000,C 180.000} C_DIS
LIN {X 29.869,Y 121.994,Z 55.077,A 180.000,B 0.000,C 180.000} C_DIS
LIN {X 29.797,Y 121.854,Z 55.073,A 180.000,B 0.000,C 180.000} C_DIS
LIN {X 29.726,Y 121.714,Z 55.070,A 180.000,B 0.000,C 180.000} C_DIS
LIN {X 29.662,Y 121.570,Z 55.066,A 180.000,B 0.000,C 180.000} C_DIS
LIN {X 29.599,Y 121.425,Z 55.062,A 180.000,B 0.000,C 180.000} C_DIS
LIN {X 29.536,Y 121.281,Z 55.059,A 180.000,B 0.000,C 180.000} C_DIS
LIN {X 29.482,Y 121.133,Z 55.056,A 180.000,B 0.000,C 180.000} C_DIS
LIN {X 29.428,Y 120.985,Z 55.052,A 180.000,B 0.000,C 180.000} C_DIS
LIN {X 29.375,Y 120.836,Z 55.049,A 180.000,B 0.000,C 180.000} C_DIS
LIN {X 29.330,Y 120.686,Z 55.046,A 180.000,B 0.000,C 180.000} C_DIS
LIN {X 29.286,Y 120.534,Z 55.043,A 180.000,B 0.000,C 180.000} C_DIS
LIN {X 29.242,Y 120.383,Z 55.040,A 180.000,B 0.000,C 180.000} C_DIS
LIN {X 29.207,Y 120.230,Z 55.037,A 180.000,B 0.000,C 180.000} C_DIS
LIN {X 29.172,Y 120.076,Z 55.034,A 180.000,B 0.000,C 180.000} C_DIS
LIN {X 29.138,Y 119.922,Z 55.032,A 180.000,B 0.000,C 180.000} C_DIS
LIN {X 29.112,Y 119.767,Z 55.029,A 180.000,B 0.000,C 180.000} C_DIS
LIN {X 29.087,Y 119.611,Z 55.027,A 180.000,B 0.000,C 180.000} C_DIS
LIN {X 29.047,Y 119.299,Z 55.022,A 180.000,B 0.000,C 180.000} C_DIS
LIN {X 29.017,Y 118.985,Z 55.018,A 180.000,B 0.000,C 180.000} C_DIS
LIN {X 29.007,Y 118.670,Z 55.014,A 180.000,B 0.000,C 180.000} C_DIS
LIN {X 29.006,Y 118.356,Z 55.011,A 180.000,B 0.000,C 180.000} C_DIS
LIN {X 29.016,Y 118.041,Z 55.008,A 180.000,B 0.000,C 180.000} C_DIS
LIN {X 29.045,Y 117.727,Z 55.005,A 180.000,B 0.000,C 180.000} C_DIS
LIN {X 29.083,Y 117.414,Z 55.003,A 180.000,B 0.000,C 180.000} C_DIS
LIN {X 29.133,Y 117.103,Z 55.002,A 180.000,B 0.000,C 180.000} C_DIS
LIN {X 29.201,Y 116.796,Z 55.001,A 180.000,B 0.000,C 180.000} C_DIS
LIN {X 29.279,Y 116.491,Z 55.000,A 180.000,B 0.000,C 180.000} C_DIS
LIN {X 29.344,Y 116.267,Z 55.000,A 180.000,B 0.000,C 180.000} C_DIS
; Cutting Move Starts
LIN {X 29.362,Y 116.204,Z 55.000,A 180.000,B 0.000,C 180.000} C_DIS
LIN {X 29.425,Y 116.025,Z 55.000,A 180.000,B 0.000,C 180.000} C_DIS
LIN {X 29.500,Y 115.816,Z 55.000,A 180.000,B 0.000,C 180.000} C_DIS
LIN {X 29.559,Y 115.667,Z 55.000,A 180.000,B 0.000,C 180.000} C_DIS
LIN {X 29.714,Y 115.310,Z 55.000,A 180.000,B 0.000,C 180.000} C_DIS
LIN {X 29.805,Y 115.131,Z 55.000,A 180.000,B 0.000,C 180.000} C_DIS
LIN {X 29.896,Y 114.952,Z 55.000,A 180.000,B 0.000,C 180.000} C_DIS
LIN {X 29.996,Y 114.774,Z 55.000,A 180.000,B 0.000,C 180.000} C_DIS
LIN {X 30.102,Y 114.595,Z 55.000,A 180.000,B 0.000,C 180.000} C_DIS
LIN {X 30.213,Y 114.416,Z 55.000,A 180.000,B 0.000,C 180.000} C_DIS
LIN {X 30.394,Y 114.150,Z 55.000,A 180.000,B 0.000,C 180.000} C_DIS
LIN {X 30.460,Y 114.058,Z 55.000,A 180.000,B 0.000,C 180.000} C_DIS
LIN {X 30.598,Y 113.880,Z 55.000,A 180.000,B 0.000,C 180.000} C_DIS
LIN {X 30.739,Y 113.701,Z 55.000,A 180.000,B 0.000,C 180.000} C_DIS
LIN {X 30.930,Y 113.484,Z 55.000,A 180.000,B 0.000,C 180.000} C_DIS
LIN {X 31.057,Y 113.343,Z 55.000,A 180.000,B 0.000,C 180.000} C_DIS
LIN {X 31.288,Y 113.112,Z 55.000,A 180.000,B 0.000,C 180.000} C_DIS
LIN {X 31.421,Y 112.986,Z 55.000,A 180.000,B 0.000,C 180.000} C_DIS
LIN {X 31.646,Y 112.788,Z 55.000,A 180.000,B 0.000,C 180.000} C_DIS
LIN {X 31.824,Y 112.641,Z 55.000,A 180.000,B 0.000,C 180.000} C_DIS
LIN {X 32.072,Y 112.450,Z 55.000,A 180.000,B 0.000,C 180.000} C_DIS
LIN {X 32.182,Y 112.373,Z 55.000,A 180.000,B 0.000,C 180.000} C_DIS
LIN {X 32.361,Y 112.251,Z 55.000,A 180.000,B 0.000,C 180.000} C_DIS
LIN {X 32.539,Y 112.135,Z 55.000,A 180.000,B 0.000,C 180.000} C_DIS
LIN {X 32.718,Y 112.029,Z 55.000,A 180.000,B 0.000,C 180.000} C_DIS
LIN {X 32.897,Y 111.924,Z 55.000,A 180.000,B 0.000,C 180.000} C_DIS
LIN {X 33.269,Y 111.734,Z 55.000,A 180.000,B 0.000,C 180.000} C_DIS
LIN {X 33.433,Y 111.660,Z 55.000,A 180.000,B 0.000,C 180.000} C_DIS
LIN {X 33.675,Y 111.556,Z 55.000,A 180.000,B 0.000,C 180.000} C_DIS
LIN {X 33.791,Y 111.509,Z 55.000,A 180.000,B 0.000,C 180.000} C_DIS
LIN {X 34.159,Y 111.377,Z 55.000,A 180.000,B 0.000,C 180.000} C_DIS
LIN {X 34.327,Y 111.326,Z 55.000,A 180.000,B 0.000,C 180.000} C_DIS
LIN {X 34.506,Y 111.274,Z 55.000,A 180.000,B 0.000,C 180.000} C_DIS
LIN {X 34.685,Y 111.226,Z 55.000,A 180.000,B 0.000,C 180.000} C_DIS
LIN {X 35.042,Y 111.146,Z 55.000,A 180.000,B 0.000,C 180.000} C_DIS
LIN {X 35.221,Y 111.114,Z 55.000,A 180.000,B 0.000,C 180.000} C_DIS
LIN {X 35.400,Y 111.086,Z 55.000,A 180.000,B 0.000,C 180.000} C_DIS
LIN {X 35.578,Y 111.059,Z 55.000,A 180.000,B 0.000,C 180.000} C_DIS
LIN {X 35.994,Y 111.019,Z 55.000,A 180.000,B 0.000,C 180.000} C_DIS
LIN {X 36.115,Y 111.013,Z 55.000,A 180.000,B 0.000,C 180.000} C_DIS
LIN {X 36.472,Y 111.002,Z 55.000,A 180.000,B 0.000,C 180.000} C_DIS
LIN {X 36.651,Y 111.006,Z 55.000,A 180.000,B 0.000,C 180.000} C_DIS
LIN {X 36.830,Y 111.012,Z 55.000,A 180.000,B 0.000,C 180.000} C_DIS
LIN {X 37.006,Y 111.019,Z 55.000,A 180.000,B 0.000,C 180.000} C_DIS
LIN {X 37.366,Y 111.053,Z 55.000,A 180.000,B 0.000,C 180.000} C_DIS
LIN {X 37.545,Y 111.077,Z 55.000,A 180.000,B 0.000,C 180.000} C_DIS
LIN {X 37.902,Y 111.134,Z 55.000,A 180.000,B 0.000,C 180.000} C_DIS
LIN {X 38.081,Y 111.173,Z 55.000,A 180.000,B 0.000,C 180.000} C_DIS
LIN {X 38.260,Y 111.213,Z 55.000,A 180.000,B 0.000,C 180.000} C_DIS
LIN {X 38.439,Y 111.258,Z 55.000,A 180.000,B 0.000,C 180.000} C_DIS
LIN {X 38.796,Y 111.362,Z 55.000,A 180.000,B 0.000,C 180.000} C_DIS
LIN {X 38.841,Y 111.377,Z 55.000,A 180.000,B 0.000,C 180.000} C_DIS
LIN {X 39.154,Y 111.489,Z 55.000,A 180.000,B 0.000,C 180.000} C_DIS
LIN {X 39.325,Y 111.556,Z 55.000,A 180.000,B 0.000,C 180.000} C_DIS
LIN {X 39.690,Y 111.714,Z 55.000,A 180.000,B 0.000,C 180.000} C_DIS
LIN {X 39.731,Y 111.734,Z 55.000,A 180.000,B 0.000,C 180.000} C_DIS
LIN {X 40.082,Y 111.913,Z 55.000,A 180.000,B 0.000,C 180.000} C_DIS
LIN {X 40.226,Y 111.996,Z 55.000,A 180.000,B 0.000,C 180.000} C_DIS
LIN {X 40.405,Y 112.102,Z 55.000,A 180.000,B 0.000,C 180.000} C_DIS
LIN {X 40.584,Y 112.213,Z 55.000,A 180.000,B 0.000,C 180.000} C_DIS
LIN {X 40.763,Y 112.335,Z 55.000,A 180.000,B 0.000,C 180.000} C_DIS
LIN {X 40.928,Y 112.450,Z 55.000,A 180.000,B 0.000,C 180.000} C_DIS
LIN {X 41.159,Y 112.628,Z 55.000,A 180.000,B 0.000,C 180.000} C_DIS
LIN {X 41.299,Y 112.739,Z 55.000,A 180.000,B 0.000,C 180.000} C_DIS
LIN {X 41.579,Y 112.986,Z 55.000,A 180.000,B 0.000,C 180.000} C_DIS
LIN {X 41.657,Y 113.057,Z 55.000,A 180.000,B 0.000,C 180.000} C_DIS
LIN {X 41.943,Y 113.343,Z 55.000,A 180.000,B 0.000,C 180.000} C_DIS
LIN {X 42.014,Y 113.421,Z 55.000,A 180.000,B 0.000,C 180.000} C_DIS
LIN {X 42.261,Y 113.701,Z 55.000,A 180.000,B 0.000,C 180.000} C_DIS
LIN {X 42.372,Y 113.841,Z 55.000,A 180.000,B 0.000,C 180.000} C_DIS
LIN {X 42.550,Y 114.072,Z 55.000,A 180.000,B 0.000,C 180.000} C_DIS
LIN {X 42.665,Y 114.237,Z 55.000,A 180.000,B 0.000,C 180.000} C_DIS
LIN {X 42.787,Y 114.416,Z 55.000,A 180.000,B 0.000,C 180.000} C_DIS
LIN {X 42.898,Y 114.595,Z 55.000,A 180.000,B 0.000,C 180.000} C_DIS
LIN {X 43.004,Y 114.774,Z 55.000,A 180.000,B 0.000,C 180.000} C_DIS
LIN {X 43.087,Y 114.918,Z 55.000,A 180.000,B 0.000,C 180.000} C_DIS
LIN {X 43.266,Y 115.269,Z 55.000,A 180.000,B 0.000,C 180.000} C_DIS
LIN {X 43.286,Y 115.310,Z 55.000,A 180.000,B 0.000,C 180.000} C_DIS
LIN {X 43.444,Y 115.675,Z 55.000,A 180.000,B 0.000,C 180.000} C_DIS
LIN {X 43.511,Y 115.846,Z 55.000,A 180.000,B 0.000,C 180.000} C_DIS
LIN {X 43.623,Y 116.159,Z 55.000,A 180.000,B 0.000,C 180.000} C_DIS
LIN {X 43.638,Y 116.204,Z 55.000,A 180.000,B 0.000,C 180.000} C_DIS
LIN {X 43.742,Y 116.561,Z 55.000,A 180.000,B 0.000,C 180.000} C_DIS
LIN {X 43.787,Y 116.740,Z 55.000,A 180.000,B 0.000,C 180.000} C_DIS
LIN {X 43.827,Y 116.919,Z 55.000,A 180.000,B 0.000,C 180.000} C_DIS
LIN {X 43.866,Y 117.098,Z 55.000,A 180.000,B 0.000,C 180.000} C_DIS
LIN {X 43.923,Y 117.455,Z 55.000,A 180.000,B 0.000,C 180.000} C_DIS
LIN {X 43.947,Y 117.634,Z 55.000,A 180.000,B 0.000,C 180.000} C_DIS
LIN {X 43.981,Y 117.994,Z 55.000,A 180.000,B 0.000,C 180.000} C_DIS
LIN {X 43.988,Y 118.170,Z 55.000,A 180.000,B 0.000,C 180.000} C_DIS
LIN {X 43.994,Y 118.349,Z 55.000,A 180.000,B 0.000,C 180.000} C_DIS
LIN {X 43.998,Y 118.528,Z 55.000,A 180.000,B 0.000,C 180.000} C_DIS
LIN {X 43.987,Y 118.885,Z 55.000,A 180.000,B 0.000,C 180.000} C_DIS
LIN {X 43.981,Y 119.006,Z 55.000,A 180.000,B 0.000,C 180.000} C_DIS
LIN {X 43.941,Y 119.422,Z 55.000,A 180.000,B 0.000,C 180.000} C_DIS
LIN {X 43.914,Y 119.600,Z 55.000,A 180.000,B 0.000,C 180.000} C_DIS
LIN {X 43.886,Y 119.779,Z 55.000,A 180.000,B 0.000,C 180.000} C_DIS
LIN {X 43.854,Y 119.958,Z 55.000,A 180.000,B 0.000,C 180.000} C_DIS
LIN {X 43.774,Y 120.315,Z 55.000,A 180.000,B 0.000,C 180.000} C_DIS
LIN {X 43.726,Y 120.494,Z 55.000,A 180.000,B 0.000,C 180.000} C_DIS
LIN {X 43.674,Y 120.673,Z 55.000,A 180.000,B 0.000,C 180.000} C_DIS
LIN {X 43.623,Y 120.841,Z 55.000,A 180.000,B 0.000,C 180.000} C_DIS
LIN {X 43.491,Y 121.209,Z 55.000,A 180.000,B 0.000,C 180.000} C_DIS
LIN {X 43.444,Y 121.325,Z 55.000,A 180.000,B 0.000,C 180.000} C_DIS
LIN {X 43.340,Y 121.567,Z 55.000,A 180.000,B 0.000,C 180.000} C_DIS
LIN {X 43.266,Y 121.731,Z 55.000,A 180.000,B 0.000,C 180.000} C_DIS
LIN {X 43.076,Y 122.103,Z 55.000,A 180.000,B 0.000,C 180.000} C_DIS
LIN {X 42.971,Y 122.282,Z 55.000,A 180.000,B 0.000,C 180.000} C_DIS
LIN {X 42.865,Y 122.461,Z 55.000,A 180.000,B 0.000,C 180.000} C_DIS
LIN {X 42.749,Y 122.639,Z 55.000,A 180.000,B 0.000,C 180.000} C_DIS
LIN {X 42.627,Y 122.818,Z 55.000,A 180.000,B 0.000,C 180.000} C_DIS
LIN {X 42.550,Y 122.928,Z 55.000,A 180.000,B 0.000,C 180.000} C_DIS
LIN {X 42.359,Y 123.176,Z 55.000,A 180.000,B 0.000,C 180.000} C_DIS
LIN {X 42.212,Y 123.354,Z 55.000,A 180.000,B 0.000,C 180.000} C_DIS
LIN {X 42.014,Y 123.579,Z 55.000,A 180.000,B 0.000,C 180.000} C_DIS
LIN {X 41.888,Y 123.712,Z 55.000,A 180.000,B 0.000,C 180.000} C_DIS
LIN {X 41.657,Y 123.943,Z 55.000,A 180.000,B 0.000,C 180.000} C_DIS
LIN {X 41.516,Y 124.070,Z 55.000,A 180.000,B 0.000,C 180.000} C_DIS
LIN {X 41.299,Y 124.261,Z 55.000,A 180.000,B 0.000,C 180.000} C_DIS
LIN {X 41.120,Y 124.402,Z 55.000,A 180.000,B 0.000,C 180.000} C_DIS
LIN {X 40.942,Y 124.540,Z 55.000,A 180.000,B 0.000,C 180.000} C_DIS
LIN {X 40.850,Y 124.606,Z 55.000,A 180.000,B 0.000,C 180.000} C_DIS
LIN {X 40.584,Y 124.787,Z 55.000,A 180.000,B 0.000,C 180.000} C_DIS
LIN {X 40.405,Y 124.898,Z 55.000,A 180.000,B 0.000,C 180.000} C_DIS
LIN {X 40.226,Y 125.004,Z 55.000,A 180.000,B 0.000,C 180.000} C_DIS
LIN {X 40.048,Y 125.104,Z 55.000,A 180.000,B 0.000,C 180.000} C_DIS
LIN {X 39.869,Y 125.195,Z 55.000,A 180.000,B 0.000,C 180.000} C_DIS
LIN {X 39.690,Y 125.286,Z 55.000,A 180.000,B 0.000,C 180.000} C_DIS
LIN {X 39.333,Y 125.441,Z 55.000,A 180.000,B 0.000,C 180.000} C_DIS
LIN {X 39.184,Y 125.500,Z 55.000,A 180.000,B 0.000,C 180.000} C_DIS
LIN {X 38.975,Y 125.575,Z 55.000,A 180.000,B 0.000,C 180.000} C_DIS
LIN {X 38.796,Y 125.638,Z 55.000,A 180.000,B 0.000,C 180.000} C_DIS
LIN {X 38.439,Y 125.742,Z 55.000,A 180.000,B 0.000,C 180.000} C_DIS
LIN {X 38.260,Y 125.787,Z 55.000,A 180.000,B 0.000,C 180.000} C_DIS
LIN {X 37.944,Y 125.857,Z 55.000,A 180.000,B 0.000,C 180.000} C_DIS
LIN {X 37.902,Y 125.866,Z 55.000,A 180.000,B 0.000,C 180.000} C_DIS
LIN {X 37.545,Y 125.923,Z 55.000,A 180.000,B 0.000,C 180.000} C_DIS
LIN {X 37.366,Y 125.947,Z 55.000,A 180.000,B 0.000,C 180.000} C_DIS
LIN {X 37.009,Y 125.980,Z 55.000,A 180.000,B 0.000,C 180.000} C_DIS
LIN {X 36.830,Y 125.988,Z 55.000,A 180.000,B 0.000,C 180.000} C_DIS
LIN {X 36.651,Y 125.994,Z 55.000,A 180.000,B 0.000,C 180.000} C_DIS
LIN {X 36.472,Y 125.998,Z 55.000,A 180.000,B 0.000,C 180.000} C_DIS
LIN {X 36.115,Y 125.987,Z 55.000,A 180.000,B 0.000,C 180.000} C_DIS
LIN {X 35.936,Y 125.975,Z 55.000,A 180.000,B 0.000,C 180.000} C_DIS
LIN {X 35.578,Y 125.941,Z 55.000,A 180.000,B 0.000,C 180.000} C_DIS
LIN {X 35.400,Y 125.914,Z 55.000,A 180.000,B 0.000,C 180.000} C_DIS
LIN {X 35.221,Y 125.886,Z 55.000,A 180.000,B 0.000,C 180.000} C_DIS
LIN {X 35.056,Y 125.857,Z 55.000,A 180.000,B 0.000,C 180.000} C_DIS
LIN {X 34.685,Y 125.774,Z 55.000,A 180.000,B 0.000,C 180.000} C_DIS
LIN {X 34.506,Y 125.726,Z 55.000,A 180.000,B 0.000,C 180.000} C_DIS
LIN {X 34.327,Y 125.674,Z 55.000,A 180.000,B 0.000,C 180.000} C_DIS
LIN {X 34.148,Y 125.619,Z 55.000,A 180.000,B 0.000,C 180.000} C_DIS
LIN {X 33.791,Y 125.491,Z 55.000,A 180.000,B 0.000,C 180.000} C_DIS
LIN {X 33.612,Y 125.417,Z 55.000,A 180.000,B 0.000,C 180.000} C_DIS
LIN {X 33.390,Y 125.321,Z 55.000,A 180.000,B 0.000,C 180.000} C_DIS
LIN {X 33.254,Y 125.258,Z 55.000,A 180.000,B 0.000,C 180.000} C_DIS
LIN {X 32.897,Y 125.076,Z 55.000,A 180.000,B 0.000,C 180.000} C_DIS
LIN {X 32.718,Y 124.971,Z 55.000,A 180.000,B 0.000,C 180.000} C_DIS
LIN {X 32.539,Y 124.865,Z 55.000,A 180.000,B 0.000,C 180.000} C_DIS
LIN {X 32.413,Y 124.785,Z 55.000,A 180.000,B 0.000,C 180.000} C_DIS
LIN {X 32.150,Y 124.606,Z 55.000,A 180.000,B 0.000,C 180.000} C_DIS
LIN {X 32.003,Y 124.497,Z 55.000,A 180.000,B 0.000,C 180.000} C_DIS
LIN {X 31.824,Y 124.359,Z 55.000,A 180.000,B 0.000,C 180.000} C_DIS
LIN {X 31.687,Y 124.248,Z 55.000,A 180.000,B 0.000,C 180.000} C_DIS
LIN {X 31.467,Y 124.055,Z 55.000,A 180.000,B 0.000,C 180.000} C_DIS
LIN {X 31.291,Y 123.891,Z 55.000,A 180.000,B 0.000,C 180.000} C_DIS
LIN {X 31.109,Y 123.709,Z 55.000,A 180.000,B 0.000,C 180.000} C_DIS
LIN {X 30.945,Y 123.533,Z 55.000,A 180.000,B 0.000,C 180.000} C_DIS
LIN {X 30.752,Y 123.313,Z 55.000,A 180.000,B 0.000,C 180.000} C_DIS
LIN {X 30.641,Y 123.176,Z 55.000,A 180.000,B 0.000,C 180.000} C_DIS
LIN {X 30.503,Y 122.997,Z 55.000,A 180.000,B 0.000,C 180.000} C_DIS
LIN {X 30.394,Y 122.850,Z 55.000,A 180.000,B 0.000,C 180.000} C_DIS
LIN {X 30.215,Y 122.587,Z 55.000,A 180.000,B 0.000,C 180.000} C_DIS
LIN {X 30.135,Y 122.461,Z 55.000,A 180.000,B 0.000,C 180.000} C_DIS
LIN {X 30.029,Y 122.282,Z 55.000,A 180.000,B 0.000,C 180.000} C_DIS
LIN {X 29.924,Y 122.103,Z 55.000,A 180.000,B 0.000,C 180.000} C_DIS
LIN {X 29.742,Y 121.746,Z 55.000,A 180.000,B 0.000,C 180.000} C_DIS
LIN {X 29.679,Y 121.610,Z 55.000,A 180.000,B 0.000,C 180.000} C_DIS
LIN {X 29.583,Y 121.388,Z 55.000,A 180.000,B 0.000,C 180.000} C_DIS
LIN {X 29.509,Y 121.209,Z 55.000,A 180.000,B 0.000,C 180.000} C_DIS
LIN {X 29.381,Y 120.852,Z 55.000,A 180.000,B 0.000,C 180.000} C_DIS
LIN {X 29.326,Y 120.673,Z 55.000,A 180.000,B 0.000,C 180.000} C_DIS
LIN {X 29.274,Y 120.494,Z 55.000,A 180.000,B 0.000,C 180.000} C_DIS
LIN {X 29.226,Y 120.315,Z 55.000,A 180.000,B 0.000,C 180.000} C_DIS
LIN {X 29.143,Y 119.944,Z 55.000,A 180.000,B 0.000,C 180.000} C_DIS
LIN {X 29.114,Y 119.779,Z 55.000,A 180.000,B 0.000,C 180.000} C_DIS
LIN {X 29.086,Y 119.600,Z 55.000,A 180.000,B 0.000,C 180.000} C_DIS
LIN {X 29.059,Y 119.422,Z 55.000,A 180.000,B 0.000,C 180.000} C_DIS
LIN {X 29.025,Y 119.064,Z 55.000,A 180.000,B 0.000,C 180.000} C_DIS
LIN {X 29.013,Y 118.885,Z 55.000,A 180.000,B 0.000,C 180.000} C_DIS
LIN {X 29.002,Y 118.528,Z 55.000,A 180.000,B 0.000,C 180.000} C_DIS
LIN {X 29.006,Y 118.349,Z 55.000,A 180.000,B 0.000,C 180.000} C_DIS
LIN {X 29.012,Y 118.170,Z 55.000,A 180.000,B 0.000,C 180.000} C_DIS
LIN {X 29.020,Y 117.991,Z 55.000,A 180.000,B 0.000,C 180.000} C_DIS
LIN {X 29.053,Y 117.634,Z 55.000,A 180.000,B 0.000,C 180.000} C_DIS
LIN {X 29.077,Y 117.455,Z 55.000,A 180.000,B 0.000,C 180.000} C_DIS
LIN {X 29.134,Y 117.098,Z 55.000,A 180.000,B 0.000,C 180.000} C_DIS
LIN {X 29.143,Y 117.056,Z 55.000,A 180.000,B 0.000,C 180.000} C_DIS
LIN {X 29.213,Y 116.740,Z 55.000,A 180.000,B 0.000,C 180.000} C_DIS
LIN {X 29.258,Y 116.561,Z 55.000,A 180.000,B 0.000,C 180.000} C_DIS
LIN {X 29.344,Y 116.267,Z 55.000,A 180.000,B 0.000,C 180.000} C_DIS
; Link Move Starts
LIN {X 29.445,Y 115.969,Z 55.000,A 180.000,B 0.000,C 180.000} C_DIS
LIN {X 29.556,Y 115.674,Z 54.999,A 180.000,B 0.000,C 180.000} C_DIS
LIN {X 29.681,Y 115.385,Z 54.998,A 180.000,B 0.000,C 180.000} C_DIS
LIN {X 29.819,Y 115.102,Z 54.996,A 180.000,B 0.000,C 180.000} C_DIS
LIN {X 29.967,Y 114.823,Z 54.994,A 180.000,B 0.000,C 180.000} C_DIS
LIN {X 30.127,Y 114.552,Z 54.991,A 180.000,B 0.000,C 180.000} C_DIS
LIN {X 30.300,Y 114.289,Z 54.988,A 180.000,B 0.000,C 180.000} C_DIS
LIN {X 30.481,Y 114.031,Z 54.985,A 180.000,B 0.000,C 180.000} C_DIS
LIN {X 30.674,Y 113.782,Z 54.981,A 180.000,B 0.000,C 180.000} C_DIS
LIN {X 30.878,Y 113.543,Z 54.977,A 180.000,B 0.000,C 180.000} C_DIS
LIN {X 31.090,Y 113.310,Z 54.972,A 180.000,B 0.000,C 180.000} C_DIS
LIN {X 31.202,Y 113.199,Z 54.969,A 180.000,B 0.000,C 180.000} C_DIS
LIN {X 31.313,Y 113.087,Z 54.967,A 180.000,B 0.000,C 180.000} C_DIS
LIN {X 31.428,Y 112.980,Z 54.964,A 180.000,B 0.000,C 180.000} C_DIS
LIN {X 31.546,Y 112.875,Z 54.961,A 180.000,B 0.000,C 180.000} C_DIS
LIN {X 31.664,Y 112.771,Z 54.959,A 180.000,B 0.000,C 180.000} C_DIS
LIN {X 31.786,Y 112.671,Z 54.956,A 180.000,B 0.000,C 180.000} C_DIS
LIN {X 31.910,Y 112.575,Z 54.952,A 180.000,B 0.000,C 180.000} C_DIS
LIN {X 32.035,Y 112.478,Z 54.949,A 180.000,B 0.000,C 180.000} C_DIS
LIN {X 32.162,Y 112.386,Z 54.946,A 180.000,B 0.000,C 180.000} C_DIS
LIN {X 32.293,Y 112.297,Z 54.943,A 180.000,B 0.000,C 180.000} C_DIS
LIN {X 32.423,Y 112.209,Z 54.939,A 180.000,B 0.000,C 180.000} C_DIS
LIN {X 32.556,Y 112.125,Z 54.936,A 180.000,B 0.000,C 180.000} C_DIS
LIN {X 32.692,Y 112.045,Z 54.932,A 180.000,B 0.000,C 180.000} C_DIS
LIN {X 32.827,Y 111.964,Z 54.928,A 180.000,B 0.000,C 180.000} C_DIS
LIN {X 32.966,Y 111.889,Z 54.925,A 180.000,B 0.000,C 180.000} C_DIS
LIN {X 33.106,Y 111.817,Z 54.921,A 180.000,B 0.000,C 180.000} C_DIS
LIN {X 33.246,Y 111.746,Z 54.917,A 180.000,B 0.000,C 180.000} C_DIS
LIN {X 33.389,Y 111.680,Z 54.913,A 180.000,B 0.000,C 180.000} C_DIS
LIN {X 33.534,Y 111.617,Z 54.909,A 180.000,B 0.000,C 180.000} C_DIS
LIN {X 33.678,Y 111.554,Z 54.905,A 180.000,B 0.000,C 180.000} C_DIS
LIN {X 33.825,Y 111.497,Z 54.900,A 180.000,B 0.000,C 180.000} C_DIS
LIN {X 33.973,Y 111.444,Z 54.896,A 180.000,B 0.000,C 180.000} C_DIS
LIN {X 34.121,Y 111.390,Z 54.892,A 180.000,B 0.000,C 180.000} C_DIS
LIN {X 34.271,Y 111.343,Z 54.887,A 180.000,B 0.000,C 180.000} C_DIS
LIN {X 34.422,Y 111.299,Z 54.883,A 180.000,B 0.000,C 180.000} C_DIS
LIN {X 34.574,Y 111.255,Z 54.878,A 180.000,B 0.000,C 180.000} C_DIS
LIN {X 34.726,Y 111.216,Z 54.873,A 180.000,B 0.000,C 180.000} C_DIS
LIN {X 34.880,Y 111.182,Z 54.869,A 180.000,B 0.000,C 180.000} C_DIS
LIN {X 35.034,Y 111.148,Z 54.864,A 180.000,B 0.000,C 180.000} C_DIS
LIN {X 35.189,Y 111.119,Z 54.859,A 180.000,B 0.000,C 180.000} C_DIS
LIN {X 35.344,Y 111.095,Z 54.854,A 180.000,B 0.000,C 180.000} C_DIS
LIN {X 35.422,Y 111.082,Z 54.851,A 180.000,B 0.000,C 180.000} C_DIS
LIN {X 35.500,Y 111.070,Z 54.849,A 180.000,B 0.000,C 180.000} C_DIS
LIN {X 35.578,Y 111.059,Z 54.846,A 180.000,B 0.000,C 180.000} C_DIS
LIN {X 35.656,Y 111.051,Z 54.844,A 180.000,B 0.000,C 180.000} C_DIS
LIN {X 35.735,Y 111.044,Z 54.841,A 180.000,B 0.000,C 180.000} C_DIS
LIN {X 35.813,Y 111.036,Z 54.839,A 180.000,B 0.000,C 180.000} C_DIS
LIN {X 35.891,Y 111.029,Z 54.836,A 180.000,B 0.000,C 180.000} C_DIS
LIN {X 35.970,Y 111.022,Z 54.833,A 180.000,B 0.000,C 180.000} C_DIS
LIN {X 36.048,Y 111.015,Z 54.831,A 180.000,B 0.000,C 180.000} C_DIS
LIN {X 36.127,Y 111.013,Z 54.828,A 180.000,B 0.000,C 180.000} C_DIS
LIN {X 36.284,Y 111.008,Z 54.823,A 180.000,B 0.000,C 180.000} C_DIS
LIN {X 36.442,Y 111.003,Z 54.817,A 180.000,B 0.000,C 180.000} C_DIS
LIN {X 36.521,Y 111.002,Z 54.815,A 180.000,B 0.000,C 180.000} C_DIS
LIN {X 36.678,Y 111.007,Z 54.809,A 180.000,B 0.000,C 180.000} C_DIS
LIN {X 36.757,Y 111.009,Z 54.806,A 180.000,B 0.000,C 180.000} C_DIS
LIN {X 36.914,Y 111.014,Z 54.801,A 180.000,B 0.000,C 180.000} C_DIS
LIN {X 36.993,Y 111.018,Z 54.798,A 180.000,B 0.000,C 180.000} C_DIS
LIN {X 37.071,Y 111.026,Z 54.796,A 180.000,B 0.000,C 180.000} C_DIS
LIN {X 37.228,Y 111.040,Z 54.790,A 180.000,B 0.000,C 180.000} C_DIS
LIN {X 37.385,Y 111.055,Z 54.785,A 180.000,B 0.000,C 180.000} C_DIS
LIN {X 37.463,Y 111.064,Z 54.782,A 180.000,B 0.000,C 180.000} C_DIS
LIN {X 37.619,Y 111.089,Z 54.776,A 180.000,B 0.000,C 180.000} C_DIS
LIN {X 37.697,Y 111.101,Z 54.774,A 180.000,B 0.000,C 180.000} C_DIS
LIN {X 37.852,Y 111.126,Z 54.768,A 180.000,B 0.000,C 180.000} C_DIS
LIN {X 37.930,Y 111.140,Z 54.765,A 180.000,B 0.000,C 180.000} C_DIS
LIN {X 38.006,Y 111.157,Z 54.763,A 180.000,B 0.000,C 180.000} C_DIS
LIN {X 38.160,Y 111.191,Z 54.757,A 180.000,B 0.000,C 180.000} C_DIS
LIN {X 38.314,Y 111.225,Z 54.752,A 180.000,B 0.000,C 180.000} C_DIS
LIN {X 38.390,Y 111.244,Z 54.749,A 180.000,B 0.000,C 180.000} C_DIS
LIN {X 38.542,Y 111.288,Z 54.743,A 180.000,B 0.000,C 180.000} C_DIS
LIN {X 38.617,Y 111.310,Z 54.741,A 180.000,B 0.000,C 180.000} C_DIS
LIN {X 38.768,Y 111.354,Z 54.735,A 180.000,B 0.000,C 180.000} C_DIS
LIN {X 38.844,Y 111.378,Z 54.732,A 180.000,B 0.000,C 180.000} C_DIS
LIN {X 38.918,Y 111.404,Z 54.730,A 180.000,B 0.000,C 180.000} C_DIS
LIN {X 39.066,Y 111.458,Z 54.724,A 180.000,B 0.000,C 180.000} C_DIS
LIN {X 39.214,Y 111.511,Z 54.719,A 180.000,B 0.000,C 180.000} C_DIS
LIN {X 39.288,Y 111.540,Z 54.716,A 180.000,B 0.000,C 180.000} C_DIS
LIN {X 39.432,Y 111.602,Z 54.710,A 180.000,B 0.000,C 180.000} C_DIS
LIN {X 39.504,Y 111.633,Z 54.708,A 180.000,B 0.000,C 180.000} C_DIS
LIN {X 39.649,Y 111.696,Z 54.702,A 180.000,B 0.000,C 180.000} C_DIS
LIN {X 39.720,Y 111.729,Z 54.699,A 180.000,B 0.000,C 180.000} C_DIS
LIN {X 39.791,Y 111.765,Z 54.697,A 180.000,B 0.000,C 180.000} C_DIS
LIN {X 39.931,Y 111.836,Z 54.691,A 180.000,B 0.000,C 180.000} C_DIS
LIN {X 40.071,Y 111.908,Z 54.686,A 180.000,B 0.000,C 180.000} C_DIS
LIN {X 40.140,Y 111.945,Z 54.683,A 180.000,B 0.000,C 180.000} C_DIS
LIN {X 40.276,Y 112.025,Z 54.677,A 180.000,B 0.000,C 180.000} C_DIS
LIN {X 40.344,Y 112.066,Z 54.675,A 180.000,B 0.000,C 180.000} C_DIS
LIN {X 40.479,Y 112.146,Z 54.669,A 180.000,B 0.000,C 180.000} C_DIS
LIN {X 40.546,Y 112.188,Z 54.666,A 180.000,B 0.000,C 180.000} C_DIS
LIN {X 40.676,Y 112.276,Z 54.661,A 180.000,B 0.000,C 180.000} C_DIS
LIN {X 40.872,Y 112.409,Z 54.653,A 180.000,B 0.000,C 180.000} C_DIS
LIN {X 40.936,Y 112.455,Z 54.650,A 180.000,B 0.000,C 180.000} C_DIS
LIN {X 41.247,Y 112.696,Z 54.636,A 180.000,B 0.000,C 180.000} C_DIS
LIN {X 41.307,Y 112.746,Z 54.633,A 180.000,B 0.000,C 180.000} C_DIS
LIN {X 41.426,Y 112.851,Z 54.628,A 180.000,B 0.000,C 180.000} C_DIS
LIN {X 41.603,Y 113.007,Z 54.620,A 180.000,B 0.000,C 180.000} C_DIS
LIN {X 41.660,Y 113.061,Z 54.617,A 180.000,B 0.000,C 180.000} C_DIS
LIN {X 41.939,Y 113.339,Z 54.603,A 180.000,B 0.000,C 180.000} C_DIS
LIN {X 41.993,Y 113.397,Z 54.600,A 180.000,B 0.000,C 180.000} C_DIS
LIN {X 42.253,Y 113.692,Z 54.587,A 180.000,B 0.000,C 180.000} C_DIS
LIN {X 42.303,Y 113.753,Z 54.584,A 180.000,B 0.000,C 180.000} C_DIS
LIN {X 42.544,Y 114.064,Z 54.570,A 180.000,B 0.000,C 180.000} C_DIS
LIN {X 42.591,Y 114.128,Z 54.567,A 180.000,B 0.000,C 180.000} C_DIS
LIN {X 42.812,Y 114.453,Z 54.554,A 180.000,B 0.000,C 180.000} C_DIS
LIN {X 42.854,Y 114.520,Z 54.551,A 180.000,B 0.000,C 180.000} C_DIS
LIN {X 43.054,Y 114.859,Z 54.537,A 180.000,B 0.000,C 180.000} C_DIS
LIN {X 43.092,Y 114.928,Z 54.534,A 180.000,B 0.000,C 180.000} C_DIS
LIN {X 43.271,Y 115.279,Z 54.521,A 180.000,B 0.000,C 180.000} C_DIS
LIN {X 43.304,Y 115.350,Z 54.518,A 180.000,B 0.000,C 180.000} C_DIS
LIN {X 43.460,Y 115.712,Z 54.504,A 180.000,B 0.000,C 180.000} C_DIS
LIN {X 43.489,Y 115.785,Z 54.501,A 180.000,B 0.000,C 180.000} C_DIS
LIN {X 43.622,Y 116.156,Z 54.488,A 180.000,B 0.000,C 180.000} C_DIS
LIN {X 43.646,Y 116.231,Z 54.485,A 180.000,B 0.000,C 180.000} C_DIS
LIN {X 43.756,Y 116.609,Z 54.471,A 180.000,B 0.000,C 180.000} C_DIS
LIN {X 43.774,Y 116.685,Z 54.468,A 180.000,B 0.000,C 180.000} C_DIS
LIN {X 43.860,Y 117.070,Z 54.455,A 180.000,B 0.000,C 180.000} C_DIS
LIN {X 43.874,Y 117.147,Z 54.452,A 180.000,B 0.000,C 180.000} C_DIS
LIN {X 43.936,Y 117.536,Z 54.438,A 180.000,B 0.000,C 180.000} C_DIS
LIN {X 43.945,Y 117.614,Z 54.435,A 180.000,B 0.000,C 180.000} C_DIS
LIN {X 43.982,Y 118.006,Z 54.422,A 180.000,B 0.000,C 180.000} C_DIS
LIN {X 43.986,Y 118.085,Z 54.419,A 180.000,B 0.000,C 180.000} C_DIS
LIN {X 43.998,Y 118.479,Z 54.405,A 180.000,B 0.000,C 180.000} C_DIS
LIN {X 43.997,Y 118.557,Z 54.402,A 180.000,B 0.000,C 180.000} C_DIS
LIN {X 43.992,Y 118.715,Z 54.397,A 180.000,B 0.000,C 180.000} C_DIS
LIN {X 43.985,Y 118.951,Z 54.389,A 180.000,B 0.000,C 180.000} C_DIS
LIN {X 43.978,Y 119.029,Z 54.386,A 180.000,B 0.000,C 180.000} C_DIS
LIN {X 43.941,Y 119.421,Z 54.372,A 180.000,B 0.000,C 180.000} C_DIS
LIN {X 43.930,Y 119.499,Z 54.369,A 180.000,B 0.000,C 180.000} C_DIS
LIN {X 43.906,Y 119.655,Z 54.364,A 180.000,B 0.000,C 180.000} C_DIS
LIN {X 43.869,Y 119.888,Z 54.356,A 180.000,B 0.000,C 180.000} C_DIS
LIN {X 43.852,Y 119.965,Z 54.353,A 180.000,B 0.000,C 180.000} C_DIS
LIN {X 43.767,Y 120.350,Z 54.339,A 180.000,B 0.000,C 180.000} C_DIS
LIN {X 43.746,Y 120.426,Z 54.336,A 180.000,B 0.000,C 180.000} C_DIS
LIN {X 43.724,Y 120.501,Z 54.334,A 180.000,B 0.000,C 180.000} C_DIS
LIN {X 43.680,Y 120.652,Z 54.328,A 180.000,B 0.000,C 180.000} C_DIS
LIN {X 43.636,Y 120.804,Z 54.323,A 180.000,B 0.000,C 180.000} C_DIS
LIN {X 43.610,Y 120.878,Z 54.320,A 180.000,B 0.000,C 180.000} C_DIS
LIN {X 43.556,Y 121.026,Z 54.314,A 180.000,B 0.000,C 180.000} C_DIS
LIN {X 43.530,Y 121.100,Z 54.312,A 180.000,B 0.000,C 180.000} C_DIS
LIN {X 43.476,Y 121.249,Z 54.306,A 180.000,B 0.000,C 180.000} C_DIS
LIN {X 43.446,Y 121.321,Z 54.303,A 180.000,B 0.000,C 180.000} C_DIS
LIN {X 43.415,Y 121.393,Z 54.301,A 180.000,B 0.000,C 180.000} C_DIS
LIN {X 43.352,Y 121.538,Z 54.295,A 180.000,B 0.000,C 180.000} C_DIS
LIN {X 43.290,Y 121.683,Z 54.290,A 180.000,B 0.000,C 180.000} C_DIS
LIN {X 43.254,Y 121.753,Z 54.287,A 180.000,B 0.000,C 180.000} C_DIS
LIN {X 43.183,Y 121.893,Z 54.281,A 180.000,B 0.000,C 180.000} C_DIS
LIN {X 43.147,Y 121.964,Z 54.279,A 180.000,B 0.000,C 180.000} C_DIS
LIN {X 43.076,Y 122.104,Z 54.273,A 180.000,B 0.000,C 180.000} C_DIS
LIN {X 43.036,Y 122.172,Z 54.270,A 180.000,B 0.000,C 180.000} C_DIS
LIN {X 42.996,Y 122.240,Z 54.268,A 180.000,B 0.000,C 180.000} C_DIS
LIN {X 42.916,Y 122.375,Z 54.262,A 180.000,B 0.000,C 180.000} C_DIS
LIN {X 42.836,Y 122.511,Z 54.257,A 180.000,B 0.000,C 180.000} C_DIS
LIN {X 42.792,Y 122.576,Z 54.254,A 180.000,B 0.000,C 180.000} C_DIS
LIN {X 42.703,Y 122.707,Z 54.248,A 180.000,B 0.000,C 180.000} C_DIS
LIN {X 42.659,Y 122.772,Z 54.246,A 180.000,B 0.000,C 180.000} C_DIS
LIN {X 42.570,Y 122.902,Z 54.240,A 180.000,B 0.000,C 180.000} C_DIS
LIN {X 42.522,Y 122.965,Z 54.237,A 180.000,B 0.000,C 180.000} C_DIS
LIN {X 42.474,Y 123.027,Z 54.235,A 180.000,B 0.000,C 180.000} C_DIS
LIN {X 42.378,Y 123.151,Z 54.229,A 180.000,B 0.000,C 180.000} C_DIS
LIN {X 42.281,Y 123.276,Z 54.224,A 180.000,B 0.000,C 180.000} C_DIS
LIN {X 42.229,Y 123.335,Z 54.221,A 180.000,B 0.000,C 180.000} C_DIS
LIN {X 42.125,Y 123.453,Z 54.215,A 180.000,B 0.000,C 180.000} C_DIS
LIN {X 42.073,Y 123.512,Z 54.213,A 180.000,B 0.000,C 180.000} C_DIS
LIN {X 41.969,Y 123.630,Z 54.207,A 180.000,B 0.000,C 180.000} C_DIS
LIN {X 41.913,Y 123.686,Z 54.204,A 180.000,B 0.000,C 180.000} C_DIS
LIN {X 41.858,Y 123.742,Z 54.202,A 180.000,B 0.000,C 180.000} C_DIS
LIN {X 41.746,Y 123.853,Z 54.196,A 180.000,B 0.000,C 180.000} C_DIS
LIN {X 41.635,Y 123.965,Z 54.191,A 180.000,B 0.000,C 180.000} C_DIS
LIN {X 41.576,Y 124.017,Z 54.188,A 180.000,B 0.000,C 180.000} C_DIS
LIN {X 41.458,Y 124.121,Z 54.182,A 180.000,B 0.000,C 180.000} C_DIS
LIN {X 41.340,Y 124.225,Z 54.177,A 180.000,B 0.000,C 180.000} C_DIS
LIN {X 41.280,Y 124.277,Z 54.174,A 180.000,B 0.000,C 180.000} C_DIS
LIN {X 41.218,Y 124.326,Z 54.172,A 180.000,B 0.000,C 180.000} C_DIS
LIN {X 41.094,Y 124.422,Z 54.166,A 180.000,B 0.000,C 180.000} C_DIS
LIN {X 41.032,Y 124.470,Z 54.164,A 180.000,B 0.000,C 180.000} C_DIS
LIN {X 40.969,Y 124.519,Z 54.161,A 180.000,B 0.000,C 180.000} C_DIS
LIN {X 40.907,Y 124.567,Z 54.159,A 180.000,B 0.000,C 180.000} C_DIS
LIN {X 40.842,Y 124.611,Z 54.156,A 180.000,B 0.000,C 180.000} C_DIS
LIN {X 40.777,Y 124.656,Z 54.154,A 180.000,B 0.000,C 180.000} C_DIS
LIN {X 40.712,Y 124.700,Z 54.151,A 180.000,B 0.000,C 180.000} C_DIS
LIN {X 40.647,Y 124.744,Z 54.149,A 180.000,B 0.000,C 180.000} C_DIS
LIN {X 40.516,Y 124.833,Z 54.144,A 180.000,B 0.000,C 180.000} C_DIS
LIN {X 40.381,Y 124.913,Z 54.139,A 180.000,B 0.000,C 180.000} C_DIS
LIN {X 40.245,Y 124.993,Z 54.134,A 180.000,B 0.000,C 180.000} C_DIS
LIN {X 40.109,Y 125.073,Z 54.129,A 180.000,B 0.000,C 180.000} C_DIS
LIN {X 39.969,Y 125.144,Z 54.124,A 180.000,B 0.000,C 180.000} C_DIS
LIN {X 39.829,Y 125.216,Z 54.120,A 180.000,B 0.000,C 180.000} C_DIS
LIN {X 39.688,Y 125.287,Z 54.115,A 180.000,B 0.000,C 180.000} C_DIS
LIN {X 39.544,Y 125.350,Z 54.111,A 180.000,B 0.000,C 180.000} C_DIS
LIN {X 39.399,Y 125.412,Z 54.106,A 180.000,B 0.000,C 180.000} C_DIS
LIN {X 39.254,Y 125.474,Z 54.102,A 180.000,B 0.000,C 180.000} C_DIS
LIN {X 39.106,Y 125.528,Z 54.097,A 180.000,B 0.000,C 180.000} C_DIS
LIN {X 38.958,Y 125.581,Z 54.093,A 180.000,B 0.000,C 180.000} C_DIS
LIN {X 38.810,Y 125.634,Z 54.089,A 180.000,B 0.000,C 180.000} C_DIS
LIN {X 38.658,Y 125.678,Z 54.085,A 180.000,B 0.000,C 180.000} C_DIS
LIN {X 38.507,Y 125.722,Z 54.081,A 180.000,B 0.000,C 180.000} C_DIS
LIN {X 38.356,Y 125.765,Z 54.077,A 180.000,B 0.000,C 180.000} C_DIS
LIN {X 38.202,Y 125.800,Z 54.073,A 180.000,B 0.000,C 180.000} C_DIS
LIN {X 38.048,Y 125.834,Z 54.070,A 180.000,B 0.000,C 180.000} C_DIS
LIN {X 37.894,Y 125.868,Z 54.066,A 180.000,B 0.000,C 180.000} C_DIS
LIN {X 37.739,Y 125.892,Z 54.062,A 180.000,B 0.000,C 180.000} C_DIS
LIN {X 37.583,Y 125.917,Z 54.059,A 180.000,B 0.000,C 180.000} C_DIS
LIN {X 37.427,Y 125.941,Z 54.056,A 180.000,B 0.000,C 180.000} C_DIS
LIN {X 37.271,Y 125.956,Z 54.052,A 180.000,B 0.000,C 180.000} C_DIS
LIN {X 37.114,Y 125.970,Z 54.049,A 180.000,B 0.000,C 180.000} C_DIS
LIN {X 36.957,Y 125.984,Z 54.046,A 180.000,B 0.000,C 180.000} C_DIS
LIN {X 36.799,Y 125.989,Z 54.043,A 180.000,B 0.000,C 180.000} C_DIS
LIN {X 36.642,Y 125.994,Z 54.040,A 180.000,B 0.000,C 180.000} C_DIS
LIN {X 36.485,Y 125.998,Z 54.037,A 180.000,B 0.000,C 180.000} C_DIS
LIN {X 36.327,Y 125.993,Z 54.034,A 180.000,B 0.000,C 180.000} C_DIS
LIN {X 36.170,Y 125.988,Z 54.032,A 180.000,B 0.000,C 180.000} C_DIS
LIN {X 36.012,Y 125.982,Z 54.029,A 180.000,B 0.000,C 180.000} C_DIS
LIN {X 35.855,Y 125.968,Z 54.027,A 180.000,B 0.000,C 180.000} C_DIS
LIN {X 35.542,Y 125.937,Z 54.022,A 180.000,B 0.000,C 180.000} C_DIS
LIN {X 35.231,Y 125.887,Z 54.018,A 180.000,B 0.000,C 180.000} C_DIS
LIN {X 34.922,Y 125.827,Z 54.014,A 180.000,B 0.000,C 180.000} C_DIS
LIN {X 34.615,Y 125.757,Z 54.011,A 180.000,B 0.000,C 180.000} C_DIS
LIN {X 34.312,Y 125.669,Z 54.008,A 180.000,B 0.000,C 180.000} C_DIS
LIN {X 34.013,Y 125.571,Z 54.005,A 180.000,B 0.000,C 180.000} C_DIS
LIN {X 33.717,Y 125.463,Z 54.003,A 180.000,B 0.000,C 180.000} C_DIS
LIN {X 33.428,Y 125.337,Z 54.002,A 180.000,B 0.000,C 180.000} C_DIS
LIN {X 33.144,Y 125.202,Z 54.001,A 180.000,B 0.000,C 180.000} C_DIS
LIN {X 32.864,Y 125.057,Z 54.000,A 180.000,B 0.000,C 180.000} C_DIS
LIN {X 32.664,Y 124.939,Z 54.000,A 180.000,B 0.000,C 180.000} C_DIS
; Cutting Move Starts
LIN {X 32.539,Y 124.865,Z 54.000,A 180.000,B 0.000,C 180.000} C_DIS
LIN {X 32.413,Y 124.785,Z 54.000,A 180.000,B 0.000,C 180.000} C_DIS
LIN {X 32.150,Y 124.606,Z 54.000,A 180.000,B 0.000,C 180.000} C_DIS
LIN {X 32.003,Y 124.497,Z 54.000,A 180.000,B 0.000,C 180.000} C_DIS
LIN {X 31.824,Y 124.359,Z 54.000,A 180.000,B 0.000,C 180.000} C_DIS
LIN {X 31.687,Y 124.248,Z 54.000,A 180.000,B 0.000,C 180.000} C_DIS
LIN {X 31.467,Y 124.055,Z 54.000,A 180.000,B 0.000,C 180.000} C_DIS
LIN {X 31.291,Y 123.891,Z 54.000,A 180.000,B 0.000,C 180.000} C_DIS
LIN {X 31.109,Y 123.709,Z 54.000,A 180.000,B 0.000,C 180.000} C_DIS
LIN {X 30.945,Y 123.533,Z 54.000,A 180.000,B 0.000,C 180.000} C_DIS
LIN {X 30.752,Y 123.313,Z 54.000,A 180.000,B 0.000,C 180.000} C_DIS
LIN {X 30.641,Y 123.176,Z 54.000,A 180.000,B 0.000,C 180.000} C_DIS
LIN {X 30.503,Y 122.997,Z 54.000,A 180.000,B 0.000,C 180.000} C_DIS
LIN {X 30.394,Y 122.850,Z 54.000,A 180.000,B 0.000,C 180.000} C_DIS
LIN {X 30.215,Y 122.587,Z 54.000,A 180.000,B 0.000,C 180.000} C_DIS
LIN {X 30.135,Y 122.461,Z 54.000,A 180.000,B 0.000,C 180.000} C_DIS
LIN {X 30.029,Y 122.282,Z 54.000,A 180.000,B 0.000,C 180.000} C_DIS
LIN {X 29.924,Y 122.103,Z 54.000,A 180.000,B 0.000,C 180.000} C_DIS
LIN {X 29.742,Y 121.746,Z 54.000,A 180.000,B 0.000,C 180.000} C_DIS
LIN {X 29.679,Y 121.610,Z 54.000,A 180.000,B 0.000,C 180.000} C_DIS
LIN {X 29.583,Y 121.388,Z 54.000,A 180.000,B 0.000,C 180.000} C_DIS
LIN {X 29.509,Y 121.209,Z 54.000,A 180.000,B 0.000,C 180.000} C_DIS
LIN {X 29.381,Y 120.852,Z 54.000,A 180.000,B 0.000,C 180.000} C_DIS
LIN {X 29.326,Y 120.673,Z 54.000,A 180.000,B 0.000,C 180.000} C_DIS
LIN {X 29.274,Y 120.494,Z 54.000,A 180.000,B 0.000,C 180.000} C_DIS
LIN {X 29.226,Y 120.315,Z 54.000,A 180.000,B 0.000,C 180.000} C_DIS
LIN {X 29.143,Y 119.944,Z 54.000,A 180.000,B 0.000,C 180.000} C_DIS
LIN {X 29.114,Y 119.779,Z 54.000,A 180.000,B 0.000,C 180.000} C_DIS
LIN {X 29.086,Y 119.600,Z 54.000,A 180.000,B 0.000,C 180.000} C_DIS
LIN {X 29.059,Y 119.422,Z 54.000,A 180.000,B 0.000,C 180.000} C_DIS
LIN {X 29.025,Y 119.064,Z 54.000,A 180.000,B 0.000,C 180.000} C_DIS
LIN {X 29.013,Y 118.885,Z 54.000,A 180.000,B 0.000,C 180.000} C_DIS
LIN {X 29.002,Y 118.528,Z 54.000,A 180.000,B 0.000,C 180.000} C_DIS
LIN {X 29.006,Y 118.349,Z 54.000,A 180.000,B 0.000,C 180.000} C_DIS
LIN {X 29.012,Y 118.170,Z 54.000,A 180.000,B 0.000,C 180.000} C_DIS
LIN {X 29.020,Y 117.991,Z 54.000,A 180.000,B 0.000,C 180.000} C_DIS
LIN {X 29.053,Y 117.634,Z 54.000,A 180.000,B 0.000,C 180.000} C_DIS
LIN {X 29.077,Y 117.455,Z 54.000,A 180.000,B 0.000,C 180.000} C_DIS
LIN {X 29.134,Y 117.098,Z 54.000,A 180.000,B 0.000,C 180.000} C_DIS
LIN {X 29.143,Y 117.056,Z 54.000,A 180.000,B 0.000,C 180.000} C_DIS
LIN {X 29.213,Y 116.740,Z 54.000,A 180.000,B 0.000,C 180.000} C_DIS
LIN {X 29.258,Y 116.561,Z 54.000,A 180.000,B 0.000,C 180.000} C_DIS
LIN {X 29.344,Y 116.267,Z 54.000,A 180.000,B 0.000,C 180.000} C_DIS
LIN {X 29.362,Y 116.204,Z 54.000,A 180.000,B 0.000,C 180.000} C_DIS
LIN {X 29.425,Y 116.025,Z 54.000,A 180.000,B 0.000,C 180.000} C_DIS
LIN {X 29.500,Y 115.816,Z 54.000,A 180.000,B 0.000,C 180.000} C_DIS
LIN {X 29.559,Y 115.667,Z 54.000,A 180.000,B 0.000,C 180.000} C_DIS
LIN {X 29.714,Y 115.310,Z 54.000,A 180.000,B 0.000,C 180.000} C_DIS
LIN {X 29.805,Y 115.131,Z 54.000,A 180.000,B 0.000,C 180.000} C_DIS
LIN {X 29.896,Y 114.952,Z 54.000,A 180.000,B 0.000,C 180.000} C_DIS
LIN {X 29.996,Y 114.774,Z 54.000,A 180.000,B 0.000,C 180.000} C_DIS
LIN {X 30.102,Y 114.595,Z 54.000,A 180.000,B 0.000,C 180.000} C_DIS
LIN {X 30.213,Y 114.416,Z 54.000,A 180.000,B 0.000,C 180.000} C_DIS
LIN {X 30.394,Y 114.150,Z 54.000,A 180.000,B 0.000,C 180.000} C_DIS
LIN {X 30.460,Y 114.058,Z 54.000,A 180.000,B 0.000,C 180.000} C_DIS
LIN {X 30.598,Y 113.880,Z 54.000,A 180.000,B 0.000,C 180.000} C_DIS
LIN {X 30.739,Y 113.701,Z 54.000,A 180.000,B 0.000,C 180.000} C_DIS
LIN {X 30.930,Y 113.484,Z 54.000,A 180.000,B 0.000,C 180.000} C_DIS
LIN {X 31.057,Y 113.343,Z 54.000,A 180.000,B 0.000,C 180.000} C_DIS
LIN {X 31.288,Y 113.112,Z 54.000,A 180.000,B 0.000,C 180.000} C_DIS
LIN {X 31.421,Y 112.986,Z 54.000,A 180.000,B 0.000,C 180.000} C_DIS
LIN {X 31.646,Y 112.788,Z 54.000,A 180.000,B 0.000,C 180.000} C_DIS
LIN {X 31.824,Y 112.641,Z 54.000,A 180.000,B 0.000,C 180.000} C_DIS
LIN {X 32.072,Y 112.450,Z 54.000,A 180.000,B 0.000,C 180.000} C_DIS
LIN {X 32.182,Y 112.373,Z 54.000,A 180.000,B 0.000,C 180.000} C_DIS
LIN {X 32.361,Y 112.251,Z 54.000,A 180.000,B 0.000,C 180.000} C_DIS
LIN {X 32.539,Y 112.135,Z 54.000,A 180.000,B 0.000,C 180.000} C_DIS
LIN {X 32.718,Y 112.029,Z 54.000,A 180.000,B 0.000,C 180.000} C_DIS
LIN {X 32.897,Y 111.924,Z 54.000,A 180.000,B 0.000,C 180.000} C_DIS
LIN {X 33.269,Y 111.734,Z 54.000,A 180.000,B 0.000,C 180.000} C_DIS
LIN {X 33.433,Y 111.660,Z 54.000,A 180.000,B 0.000,C 180.000} C_DIS
LIN {X 33.675,Y 111.556,Z 54.000,A 180.000,B 0.000,C 180.000} C_DIS
LIN {X 33.791,Y 111.509,Z 54.000,A 180.000,B 0.000,C 180.000} C_DIS
LIN {X 34.159,Y 111.377,Z 54.000,A 180.000,B 0.000,C 180.000} C_DIS
LIN {X 34.327,Y 111.326,Z 54.000,A 180.000,B 0.000,C 180.000} C_DIS
LIN {X 34.506,Y 111.274,Z 54.000,A 180.000,B 0.000,C 180.000} C_DIS
LIN {X 34.685,Y 111.226,Z 54.000,A 180.000,B 0.000,C 180.000} C_DIS
LIN {X 35.042,Y 111.146,Z 54.000,A 180.000,B 0.000,C 180.000} C_DIS
LIN {X 35.221,Y 111.114,Z 54.000,A 180.000,B 0.000,C 180.000} C_DIS
LIN {X 35.400,Y 111.086,Z 54.000,A 180.000,B 0.000,C 180.000} C_DIS
LIN {X 35.578,Y 111.059,Z 54.000,A 180.000,B 0.000,C 180.000} C_DIS
LIN {X 35.994,Y 111.019,Z 54.000,A 180.000,B 0.000,C 180.000} C_DIS
LIN {X 36.115,Y 111.013,Z 54.000,A 180.000,B 0.000,C 180.000} C_DIS
LIN {X 36.472,Y 111.002,Z 54.000,A 180.000,B 0.000,C 180.000} C_DIS
LIN {X 36.651,Y 111.006,Z 54.000,A 180.000,B 0.000,C 180.000} C_DIS
LIN {X 36.830,Y 111.012,Z 54.000,A 180.000,B 0.000,C 180.000} C_DIS
LIN {X 37.006,Y 111.019,Z 54.000,A 180.000,B 0.000,C 180.000} C_DIS
LIN {X 37.366,Y 111.053,Z 54.000,A 180.000,B 0.000,C 180.000} C_DIS
LIN {X 37.545,Y 111.077,Z 54.000,A 180.000,B 0.000,C 180.000} C_DIS
LIN {X 37.902,Y 111.134,Z 54.000,A 180.000,B 0.000,C 180.000} C_DIS
LIN {X 38.081,Y 111.173,Z 54.000,A 180.000,B 0.000,C 180.000} C_DIS
LIN {X 38.260,Y 111.213,Z 54.000,A 180.000,B 0.000,C 180.000} C_DIS
LIN {X 38.439,Y 111.258,Z 54.000,A 180.000,B 0.000,C 180.000} C_DIS
LIN {X 38.796,Y 111.362,Z 54.000,A 180.000,B 0.000,C 180.000} C_DIS
LIN {X 38.841,Y 111.377,Z 54.000,A 180.000,B 0.000,C 180.000} C_DIS
LIN {X 39.154,Y 111.489,Z 54.000,A 180.000,B 0.000,C 180.000} C_DIS
LIN {X 39.325,Y 111.556,Z 54.000,A 180.000,B 0.000,C 180.000} C_DIS
LIN {X 39.690,Y 111.714,Z 54.000,A 180.000,B 0.000,C 180.000} C_DIS
LIN {X 39.731,Y 111.734,Z 54.000,A 180.000,B 0.000,C 180.000} C_DIS
LIN {X 40.082,Y 111.913,Z 54.000,A 180.000,B 0.000,C 180.000} C_DIS
LIN {X 40.226,Y 111.996,Z 54.000,A 180.000,B 0.000,C 180.000} C_DIS
LIN {X 40.405,Y 112.102,Z 54.000,A 180.000,B 0.000,C 180.000} C_DIS
LIN {X 40.584,Y 112.213,Z 54.000,A 180.000,B 0.000,C 180.000} C_DIS
LIN {X 40.763,Y 112.335,Z 54.000,A 180.000,B 0.000,C 180.000} C_DIS
LIN {X 40.928,Y 112.450,Z 54.000,A 180.000,B 0.000,C 180.000} C_DIS
LIN {X 41.159,Y 112.628,Z 54.000,A 180.000,B 0.000,C 180.000} C_DIS
LIN {X 41.299,Y 112.739,Z 54.000,A 180.000,B 0.000,C 180.000} C_DIS
LIN {X 41.579,Y 112.986,Z 54.000,A 180.000,B 0.000,C 180.000} C_DIS
LIN {X 41.657,Y 113.057,Z 54.000,A 180.000,B 0.000,C 180.000} C_DIS
LIN {X 41.943,Y 113.343,Z 54.000,A 180.000,B 0.000,C 180.000} C_DIS
LIN {X 42.014,Y 113.421,Z 54.000,A 180.000,B 0.000,C 180.000} C_DIS
LIN {X 42.261,Y 113.701,Z 54.000,A 180.000,B 0.000,C 180.000} C_DIS
LIN {X 42.372,Y 113.841,Z 54.000,A 180.000,B 0.000,C 180.000} C_DIS
LIN {X 42.550,Y 114.072,Z 54.000,A 180.000,B 0.000,C 180.000} C_DIS
LIN {X 42.665,Y 114.237,Z 54.000,A 180.000,B 0.000,C 180.000} C_DIS
LIN {X 42.787,Y 114.416,Z 54.000,A 180.000,B 0.000,C 180.000} C_DIS
LIN {X 42.898,Y 114.595,Z 54.000,A 180.000,B 0.000,C 180.000} C_DIS
LIN {X 43.004,Y 114.774,Z 54.000,A 180.000,B 0.000,C 180.000} C_DIS
LIN {X 43.087,Y 114.918,Z 54.000,A 180.000,B 0.000,C 180.000} C_DIS
LIN {X 43.266,Y 115.269,Z 54.000,A 180.000,B 0.000,C 180.000} C_DIS
LIN {X 43.286,Y 115.310,Z 54.000,A 180.000,B 0.000,C 180.000} C_DIS
LIN {X 43.444,Y 115.675,Z 54.000,A 180.000,B 0.000,C 180.000} C_DIS
LIN {X 43.511,Y 115.846,Z 54.000,A 180.000,B 0.000,C 180.000} C_DIS
LIN {X 43.623,Y 116.159,Z 54.000,A 180.000,B 0.000,C 180.000} C_DIS
LIN {X 43.638,Y 116.204,Z 54.000,A 180.000,B 0.000,C 180.000} C_DIS
LIN {X 43.742,Y 116.561,Z 54.000,A 180.000,B 0.000,C 180.000} C_DIS
LIN {X 43.787,Y 116.740,Z 54.000,A 180.000,B 0.000,C 180.000} C_DIS
LIN {X 43.827,Y 116.919,Z 54.000,A 180.000,B 0.000,C 180.000} C_DIS
LIN {X 43.866,Y 117.098,Z 54.000,A 180.000,B 0.000,C 180.000} C_DIS
LIN {X 43.923,Y 117.455,Z 54.000,A 180.000,B 0.000,C 180.000} C_DIS
LIN {X 43.947,Y 117.634,Z 54.000,A 180.000,B 0.000,C 180.000} C_DIS
LIN {X 43.981,Y 117.994,Z 54.000,A 180.000,B 0.000,C 180.000} C_DIS
LIN {X 43.988,Y 118.170,Z 54.000,A 180.000,B 0.000,C 180.000} C_DIS
LIN {X 43.994,Y 118.349,Z 54.000,A 180.000,B 0.000,C 180.000} C_DIS
LIN {X 43.998,Y 118.528,Z 54.000,A 180.000,B 0.000,C 180.000} C_DIS
LIN {X 43.987,Y 118.885,Z 54.000,A 180.000,B 0.000,C 180.000} C_DIS
LIN {X 43.981,Y 119.006,Z 54.000,A 180.000,B 0.000,C 180.000} C_DIS
LIN {X 43.941,Y 119.422,Z 54.000,A 180.000,B 0.000,C 180.000} C_DIS
LIN {X 43.914,Y 119.600,Z 54.000,A 180.000,B 0.000,C 180.000} C_DIS
LIN {X 43.886,Y 119.779,Z 54.000,A 180.000,B 0.000,C 180.000} C_DIS
LIN {X 43.854,Y 119.958,Z 54.000,A 180.000,B 0.000,C 180.000} C_DIS
LIN {X 43.774,Y 120.315,Z 54.000,A 180.000,B 0.000,C 180.000} C_DIS
LIN {X 43.726,Y 120.494,Z 54.000,A 180.000,B 0.000,C 180.000} C_DIS
LIN {X 43.674,Y 120.673,Z 54.000,A 180.000,B 0.000,C 180.000} C_DIS
LIN {X 43.623,Y 120.841,Z 54.000,A 180.000,B 0.000,C 180.000} C_DIS
LIN {X 43.491,Y 121.209,Z 54.000,A 180.000,B 0.000,C 180.000} C_DIS
LIN {X 43.444,Y 121.325,Z 54.000,A 180.000,B 0.000,C 180.000} C_DIS
LIN {X 43.340,Y 121.567,Z 54.000,A 180.000,B 0.000,C 180.000} C_DIS
LIN {X 43.266,Y 121.731,Z 54.000,A 180.000,B 0.000,C 180.000} C_DIS
LIN {X 43.076,Y 122.103,Z 54.000,A 180.000,B 0.000,C 180.000} C_DIS
LIN {X 42.971,Y 122.282,Z 54.000,A 180.000,B 0.000,C 180.000} C_DIS
LIN {X 42.865,Y 122.461,Z 54.000,A 180.000,B 0.000,C 180.000} C_DIS
LIN {X 42.749,Y 122.639,Z 54.000,A 180.000,B 0.000,C 180.000} C_DIS
LIN {X 42.627,Y 122.818,Z 54.000,A 180.000,B 0.000,C 180.000} C_DIS
LIN {X 42.550,Y 122.928,Z 54.000,A 180.000,B 0.000,C 180.000} C_DIS
LIN {X 42.359,Y 123.176,Z 54.000,A 180.000,B 0.000,C 180.000} C_DIS
LIN {X 42.212,Y 123.354,Z 54.000,A 180.000,B 0.000,C 180.000} C_DIS
LIN {X 42.014,Y 123.579,Z 54.000,A 180.000,B 0.000,C 180.000} C_DIS
LIN {X 41.888,Y 123.712,Z 54.000,A 180.000,B 0.000,C 180.000} C_DIS
LIN {X 41.657,Y 123.943,Z 54.000,A 180.000,B 0.000,C 180.000} C_DIS
LIN {X 41.516,Y 124.070,Z 54.000,A 180.000,B 0.000,C 180.000} C_DIS
LIN {X 41.299,Y 124.261,Z 54.000,A 180.000,B 0.000,C 180.000} C_DIS
LIN {X 41.120,Y 124.402,Z 54.000,A 180.000,B 0.000,C 180.000} C_DIS
LIN {X 40.942,Y 124.540,Z 54.000,A 180.000,B 0.000,C 180.000} C_DIS
LIN {X 40.850,Y 124.606,Z 54.000,A 180.000,B 0.000,C 180.000} C_DIS
LIN {X 40.584,Y 124.787,Z 54.000,A 180.000,B 0.000,C 180.000} C_DIS
LIN {X 40.405,Y 124.898,Z 54.000,A 180.000,B 0.000,C 180.000} C_DIS
LIN {X 40.226,Y 125.004,Z 54.000,A 180.000,B 0.000,C 180.000} C_DIS
LIN {X 40.048,Y 125.104,Z 54.000,A 180.000,B 0.000,C 180.000} C_DIS
LIN {X 39.869,Y 125.195,Z 54.000,A 180.000,B 0.000,C 180.000} C_DIS
LIN {X 39.690,Y 125.286,Z 54.000,A 180.000,B 0.000,C 180.000} C_DIS
LIN {X 39.333,Y 125.441,Z 54.000,A 180.000,B 0.000,C 180.000} C_DIS
LIN {X 39.184,Y 125.500,Z 54.000,A 180.000,B 0.000,C 180.000} C_DIS
LIN {X 38.975,Y 125.575,Z 54.000,A 180.000,B 0.000,C 180.000} C_DIS
LIN {X 38.796,Y 125.638,Z 54.000,A 180.000,B 0.000,C 180.000} C_DIS
LIN {X 38.439,Y 125.742,Z 54.000,A 180.000,B 0.000,C 180.000} C_DIS
LIN {X 38.260,Y 125.787,Z 54.000,A 180.000,B 0.000,C 180.000} C_DIS
LIN {X 37.944,Y 125.857,Z 54.000,A 180.000,B 0.000,C 180.000} C_DIS
LIN {X 37.902,Y 125.866,Z 54.000,A 180.000,B 0.000,C 180.000} C_DIS
LIN {X 37.545,Y 125.923,Z 54.000,A 180.000,B 0.000,C 180.000} C_DIS
LIN {X 37.366,Y 125.947,Z 54.000,A 180.000,B 0.000,C 180.000} C_DIS
LIN {X 37.009,Y 125.980,Z 54.000,A 180.000,B 0.000,C 180.000} C_DIS
LIN {X 36.830,Y 125.988,Z 54.000,A 180.000,B 0.000,C 180.000} C_DIS
LIN {X 36.651,Y 125.994,Z 54.000,A 180.000,B 0.000,C 180.000} C_DIS
LIN {X 36.472,Y 125.998,Z 54.000,A 180.000,B 0.000,C 180.000} C_DIS
LIN {X 36.115,Y 125.987,Z 54.000,A 180.000,B 0.000,C 180.000} C_DIS
LIN {X 35.936,Y 125.975,Z 54.000,A 180.000,B 0.000,C 180.000} C_DIS
LIN {X 35.578,Y 125.941,Z 54.000,A 180.000,B 0.000,C 180.000} C_DIS
LIN {X 35.400,Y 125.914,Z 54.000,A 180.000,B 0.000,C 180.000} C_DIS
LIN {X 35.221,Y 125.886,Z 54.000,A 180.000,B 0.000,C 180.000} C_DIS
LIN {X 35.056,Y 125.857,Z 54.000,A 180.000,B 0.000,C 180.000} C_DIS
LIN {X 34.685,Y 125.774,Z 54.000,A 180.000,B 0.000,C 180.000} C_DIS
LIN {X 34.506,Y 125.726,Z 54.000,A 180.000,B 0.000,C 180.000} C_DIS
LIN {X 34.327,Y 125.674,Z 54.000,A 180.000,B 0.000,C 180.000} C_DIS
LIN {X 34.148,Y 125.619,Z 54.000,A 180.000,B 0.000,C 180.000} C_DIS
LIN {X 33.791,Y 125.491,Z 54.000,A 180.000,B 0.000,C 180.000} C_DIS
LIN {X 33.612,Y 125.417,Z 54.000,A 180.000,B 0.000,C 180.000} C_DIS
LIN {X 33.390,Y 125.321,Z 54.000,A 180.000,B 0.000,C 180.000} C_DIS
LIN {X 33.254,Y 125.258,Z 54.000,A 180.000,B 0.000,C 180.000} C_DIS
LIN {X 32.897,Y 125.076,Z 54.000,A 180.000,B 0.000,C 180.000} C_DIS
LIN {X 32.718,Y 124.971,Z 54.000,A 180.000,B 0.000,C 180.000} C_DIS
LIN {X 32.664,Y 124.939,Z 54.000,A 180.000,B 0.000,C 180.000} C_DIS
; Link Move Starts
LIN {X 32.396,Y 124.773,Z 54.000,A 180.000,B 0.000,C 180.000} C_DIS
LIN {X 32.136,Y 124.596,Z 53.999,A 180.000,B 0.000,C 180.000} C_DIS
LIN {X 31.885,Y 124.406,Z 53.998,A 180.000,B 0.000,C 180.000} C_DIS
LIN {X 31.640,Y 124.207,Z 53.996,A 180.000,B 0.000,C 180.000} C_DIS
LIN {X 31.404,Y 123.999,Z 53.994,A 180.000,B 0.000,C 180.000} C_DIS
LIN {X 31.179,Y 123.778,Z 53.991,A 180.000,B 0.000,C 180.000} C_DIS
LIN {X 30.961,Y 123.551,Z 53.988,A 180.000,B 0.000,C 180.000} C_DIS
LIN {X 30.753,Y 123.315,Z 53.985,A 180.000,B 0.000,C 180.000} C_DIS
LIN {X 30.557,Y 123.068,Z 53.981,A 180.000,B 0.000,C 180.000} C_DIS
LIN {X 30.370,Y 122.814,Z 53.977,A 180.000,B 0.000,C 180.000} C_DIS
LIN {X 30.193,Y 122.554,Z 53.972,A 180.000,B 0.000,C 180.000} C_DIS
LIN {X 30.110,Y 122.420,Z 53.969,A 180.000,B 0.000,C 180.000} C_DIS
LIN {X 30.030,Y 122.284,Z 53.967,A 180.000,B 0.000,C 180.000} C_DIS
LIN {X 29.950,Y 122.149,Z 53.964,A 180.000,B 0.000,C 180.000} C_DIS
LIN {X 29.876,Y 122.009,Z 53.961,A 180.000,B 0.000,C 180.000} C_DIS
LIN {X 29.805,Y 121.869,Z 53.959,A 180.000,B 0.000,C 180.000} C_DIS
LIN {X 29.733,Y 121.729,Z 53.956,A 180.000,B 0.000,C 180.000} C_DIS
LIN {X 29.668,Y 121.585,Z 53.952,A 180.000,B 0.000,C 180.000} C_DIS
LIN {X 29.606,Y 121.441,Z 53.949,A 180.000,B 0.000,C 180.000} C_DIS
LIN {X 29.543,Y 121.296,Z 53.946,A 180.000,B 0.000,C 180.000} C_DIS
LIN {X 29.488,Y 121.149,Z 53.943,A 180.000,B 0.000,C 180.000} C_DIS
LIN {X 29.434,Y 121.001,Z 53.939,A 180.000,B 0.000,C 180.000} C_DIS
LIN {X 29.381,Y 120.852,Z 53.936,A 180.000,B 0.000,C 180.000} C_DIS
LIN {X 29.335,Y 120.702,Z 53.932,A 180.000,B 0.000,C 180.000} C_DIS
LIN {X 29.291,Y 120.551,Z 53.928,A 180.000,B 0.000,C 180.000} C_DIS
LIN {X 29.247,Y 120.399,Z 53.925,A 180.000,B 0.000,C 180.000} C_DIS
LIN {X 29.210,Y 120.246,Z 53.921,A 180.000,B 0.000,C 180.000} C_DIS
LIN {X 29.176,Y 120.092,Z 53.917,A 180.000,B 0.000,C 180.000} C_DIS
LIN {X 29.142,Y 119.939,Z 53.913,A 180.000,B 0.000,C 180.000} C_DIS
LIN {X 29.115,Y 119.784,Z 53.909,A 180.000,B 0.000,C 180.000} C_DIS
LIN {X 29.090,Y 119.628,Z 53.905,A 180.000,B 0.000,C 180.000} C_DIS
LIN {X 29.066,Y 119.472,Z 53.900,A 180.000,B 0.000,C 180.000} C_DIS
LIN {X 29.049,Y 119.316,Z 53.896,A 180.000,B 0.000,C 180.000} C_DIS
LIN {X 29.034,Y 119.159,Z 53.892,A 180.000,B 0.000,C 180.000} C_DIS
LIN {X 29.019,Y 119.002,Z 53.887,A 180.000,B 0.000,C 180.000} C_DIS
LIN {X 29.012,Y 118.845,Z 53.883,A 180.000,B 0.000,C 180.000} C_DIS
LIN {X 29.007,Y 118.687,Z 53.878,A 180.000,B 0.000,C 180.000} C_DIS
LIN {X 29.002,Y 118.530,Z 53.873,A 180.000,B 0.000,C 180.000} C_DIS
LIN {X 29.005,Y 118.373,Z 53.869,A 180.000,B 0.000,C 180.000} C_DIS
LIN {X 29.010,Y 118.215,Z 53.864,A 180.000,B 0.000,C 180.000} C_DIS
LIN {X 29.015,Y 118.058,Z 53.859,A 180.000,B 0.000,C 180.000} C_DIS
LIN {X 29.028,Y 117.901,Z 53.854,A 180.000,B 0.000,C 180.000} C_DIS
LIN {X 29.036,Y 117.822,Z 53.851,A 180.000,B 0.000,C 180.000} C_DIS
LIN {X 29.043,Y 117.744,Z 53.849,A 180.000,B 0.000,C 180.000} C_DIS
LIN {X 29.050,Y 117.666,Z 53.846,A 180.000,B 0.000,C 180.000} C_DIS
LIN {X 29.058,Y 117.587,Z 53.844,A 180.000,B 0.000,C 180.000} C_DIS
LIN {X 29.068,Y 117.509,Z 53.841,A 180.000,B 0.000,C 180.000} C_DIS
LIN {X 29.081,Y 117.431,Z 53.839,A 180.000,B 0.000,C 180.000} C_DIS
LIN {X 29.093,Y 117.353,Z 53.836,A 180.000,B 0.000,C 180.000} C_DIS
LIN {X 29.118,Y 117.198,Z 53.831,A 180.000,B 0.000,C 180.000} C_DIS
LIN {X 29.130,Y 117.120,Z 53.828,A 180.000,B 0.000,C 180.000} C_DIS
LIN {X 29.146,Y 117.043,Z 53.825,A 180.000,B 0.000,C 180.000} C_DIS
LIN {X 29.180,Y 116.889,Z 53.820,A 180.000,B 0.000,C 180.000} C_DIS
LIN {X 29.214,Y 116.736,Z 53.815,A 180.000,B 0.000,C 180.000} C_DIS
LIN {X 29.232,Y 116.659,Z 53.812,A 180.000,B 0.000,C 180.000} C_DIS
LIN {X 29.252,Y 116.583,Z 53.809,A 180.000,B 0.000,C 180.000} C_DIS
LIN {X 29.274,Y 116.507,Z 53.806,A 180.000,B 0.000,C 180.000} C_DIS
LIN {X 29.318,Y 116.356,Z 53.801,A 180.000,B 0.000,C 180.000} C_DIS
LIN {X 29.362,Y 116.205,Z 53.796,A 180.000,B 0.000,C 180.000} C_DIS
LIN {X 29.387,Y 116.130,Z 53.793,A 180.000,B 0.000,C 180.000} C_DIS
LIN {X 29.441,Y 115.982,Z 53.787,A 180.000,B 0.000,C 180.000} C_DIS
LIN {X 29.467,Y 115.908,Z 53.785,A 180.000,B 0.000,C 180.000} C_DIS
LIN {X 29.521,Y 115.759,Z 53.779,A 180.000,B 0.000,C 180.000} C_DIS
LIN {X 29.551,Y 115.687,Z 53.776,A 180.000,B 0.000,C 180.000} C_DIS
LIN {X 29.582,Y 115.614,Z 53.774,A 180.000,B 0.000,C 180.000} C_DIS
LIN {X 29.645,Y 115.470,Z 53.768,A 180.000,B 0.000,C 180.000} C_DIS
LIN {X 29.707,Y 115.325,Z 53.763,A 180.000,B 0.000,C 180.000} C_DIS
LIN {X 29.742,Y 115.255,Z 53.760,A 180.000,B 0.000,C 180.000} C_DIS
LIN {X 29.813,Y 115.114,Z 53.754,A 180.000,B 0.000,C 180.000} C_DIS
LIN {X 29.849,Y 115.044,Z 53.752,A 180.000,B 0.000,C 180.000} C_DIS
LIN {X 29.920,Y 114.904,Z 53.746,A 180.000,B 0.000,C 180.000} C_DIS
LIN {X 29.960,Y 114.835,Z 53.743,A 180.000,B 0.000,C 180.000} C_DIS
LIN {X 30.000,Y 114.768,Z 53.741,A 180.000,B 0.000,C 180.000} C_DIS
LIN {X 30.080,Y 114.632,Z 53.735,A 180.000,B 0.000,C 180.000} C_DIS
LIN {X 30.160,Y 114.496,Z 53.730,A 180.000,B 0.000,C 180.000} C_DIS
LIN {X 30.203,Y 114.431,Z 53.727,A 180.000,B 0.000,C 180.000} C_DIS
LIN {X 30.292,Y 114.300,Z 53.721,A 180.000,B 0.000,C 180.000} C_DIS
LIN {X 30.336,Y 114.235,Z 53.719,A 180.000,B 0.000,C 180.000} C_DIS
LIN {X 30.425,Y 114.105,Z 53.713,A 180.000,B 0.000,C 180.000} C_DIS
LIN {X 30.472,Y 114.042,Z 53.710,A 180.000,B 0.000,C 180.000} C_DIS
LIN {X 30.521,Y 113.980,Z 53.708,A 180.000,B 0.000,C 180.000} C_DIS
LIN {X 30.617,Y 113.855,Z 53.702,A 180.000,B 0.000,C 180.000} C_DIS
LIN {X 30.714,Y 113.731,Z 53.697,A 180.000,B 0.000,C 180.000} C_DIS
LIN {X 30.765,Y 113.671,Z 53.694,A 180.000,B 0.000,C 180.000} C_DIS
LIN {X 30.869,Y 113.553,Z 53.688,A 180.000,B 0.000,C 180.000} C_DIS
LIN {X 30.921,Y 113.494,Z 53.686,A 180.000,B 0.000,C 180.000} C_DIS
LIN {X 31.025,Y 113.376,Z 53.680,A 180.000,B 0.000,C 180.000} C_DIS
LIN {X 31.081,Y 113.320,Z 53.677,A 180.000,B 0.000,C 180.000} C_DIS
LIN {X 31.192,Y 113.208,Z 53.672,A 180.000,B 0.000,C 180.000} C_DIS
LIN {X 31.303,Y 113.097,Z 53.666,A 180.000,B 0.000,C 180.000} C_DIS
LIN {X 31.359,Y 113.041,Z 53.664,A 180.000,B 0.000,C 180.000} C_DIS
LIN {X 31.418,Y 112.989,Z 53.661,A 180.000,B 0.000,C 180.000} C_DIS
LIN {X 31.713,Y 112.728,Z 53.647,A 180.000,B 0.000,C 180.000} C_DIS
LIN {X 31.775,Y 112.680,Z 53.644,A 180.000,B 0.000,C 180.000} C_DIS
LIN {X 31.899,Y 112.583,Z 53.639,A 180.000,B 0.000,C 180.000} C_DIS
LIN {X 32.086,Y 112.438,Z 53.631,A 180.000,B 0.000,C 180.000} C_DIS
LIN {X 32.151,Y 112.394,Z 53.628,A 180.000,B 0.000,C 180.000} C_DIS
LIN {X 32.477,Y 112.172,Z 53.614,A 180.000,B 0.000,C 180.000} C_DIS
LIN {X 32.544,Y 112.132,Z 53.611,A 180.000,B 0.000,C 180.000} C_DIS
LIN {X 32.748,Y 112.011,Z 53.603,A 180.000,B 0.000,C 180.000} C_DIS
LIN {X 32.883,Y 111.931,Z 53.598,A 180.000,B 0.000,C 180.000} C_DIS
LIN {X 32.953,Y 111.895,Z 53.595,A 180.000,B 0.000,C 180.000} C_DIS
LIN {X 33.304,Y 111.716,Z 53.581,A 180.000,B 0.000,C 180.000} C_DIS
LIN {X 33.376,Y 111.685,Z 53.578,A 180.000,B 0.000,C 180.000} C_DIS
LIN {X 33.738,Y 111.529,Z 53.565,A 180.000,B 0.000,C 180.000} C_DIS
LIN {X 33.812,Y 111.502,Z 53.562,A 180.000,B 0.000,C 180.000} C_DIS
LIN {X 34.182,Y 111.368,Z 53.548,A 180.000,B 0.000,C 180.000} C_DIS
LIN {X 34.258,Y 111.346,Z 53.545,A 180.000,B 0.000,C 180.000} C_DIS
LIN {X 34.560,Y 111.259,Z 53.534,A 180.000,B 0.000,C 180.000} C_DIS
LIN {X 34.636,Y 111.237,Z 53.532,A 180.000,B 0.000,C 180.000} C_DIS
LIN {X 35.020,Y 111.151,Z 53.518,A 180.000,B 0.000,C 180.000} C_DIS
LIN {X 35.097,Y 111.134,Z 53.515,A 180.000,B 0.000,C 180.000} C_DIS
LIN {X 35.486,Y 111.072,Z 53.501,A 180.000,B 0.000,C 180.000} C_DIS
LIN {X 35.564,Y 111.060,Z 53.499,A 180.000,B 0.000,C 180.000} C_DIS
LIN {X 35.956,Y 111.023,Z 53.485,A 180.000,B 0.000,C 180.000} C_DIS
LIN {X 36.035,Y 111.016,Z 53.482,A 180.000,B 0.000,C 180.000} C_DIS
LIN {X 36.428,Y 111.003,Z 53.468,A 180.000,B 0.000,C 180.000} C_DIS
LIN {X 36.507,Y 111.001,Z 53.466,A 180.000,B 0.000,C 180.000} C_DIS
LIN {X 36.900,Y 111.014,Z 53.452,A 180.000,B 0.000,C 180.000} C_DIS
LIN {X 36.979,Y 111.017,Z 53.449,A 180.000,B 0.000,C 180.000} C_DIS
LIN {X 37.371,Y 111.054,Z 53.435,A 180.000,B 0.000,C 180.000} C_DIS
LIN {X 37.450,Y 111.062,Z 53.433,A 180.000,B 0.000,C 180.000} C_DIS
LIN {X 37.838,Y 111.123,Z 53.419,A 180.000,B 0.000,C 180.000} C_DIS
LIN {X 37.916,Y 111.137,Z 53.416,A 180.000,B 0.000,C 180.000} C_DIS
LIN {X 38.300,Y 111.222,Z 53.402,A 180.000,B 0.000,C 180.000} C_DIS
LIN {X 38.377,Y 111.240,Z 53.400,A 180.000,B 0.000,C 180.000} C_DIS
LIN {X 38.604,Y 111.306,Z 53.391,A 180.000,B 0.000,C 180.000} C_DIS
LIN {X 38.755,Y 111.350,Z 53.386,A 180.000,B 0.000,C 180.000} C_DIS
LIN {X 38.831,Y 111.373,Z 53.383,A 180.000,B 0.000,C 180.000} C_DIS
LIN {X 39.201,Y 111.506,Z 53.369,A 180.000,B 0.000,C 180.000} C_DIS
LIN {X 39.275,Y 111.534,Z 53.367,A 180.000,B 0.000,C 180.000} C_DIS
LIN {X 39.492,Y 111.628,Z 53.358,A 180.000,B 0.000,C 180.000} C_DIS
LIN {X 39.636,Y 111.690,Z 53.353,A 180.000,B 0.000,C 180.000} C_DIS
LIN {X 39.708,Y 111.723,Z 53.350,A 180.000,B 0.000,C 180.000} C_DIS
LIN {X 40.059,Y 111.901,Z 53.336,A 180.000,B 0.000,C 180.000} C_DIS
LIN {X 40.129,Y 111.938,Z 53.334,A 180.000,B 0.000,C 180.000} C_DIS
LIN {X 40.264,Y 112.018,Z 53.328,A 180.000,B 0.000,C 180.000} C_DIS
LIN {X 40.467,Y 112.139,Z 53.320,A 180.000,B 0.000,C 180.000} C_DIS
LIN {X 40.535,Y 112.180,Z 53.317,A 180.000,B 0.000,C 180.000} C_DIS
LIN {X 40.860,Y 112.401,Z 53.303,A 180.000,B 0.000,C 180.000} C_DIS
LIN {X 40.925,Y 112.447,Z 53.301,A 180.000,B 0.000,C 180.000} C_DIS
LIN {X 41.049,Y 112.543,Z 53.295,A 180.000,B 0.000,C 180.000} C_DIS
LIN {X 41.236,Y 112.688,Z 53.287,A 180.000,B 0.000,C 180.000} C_DIS
LIN {X 41.297,Y 112.737,Z 53.284,A 180.000,B 0.000,C 180.000} C_DIS
LIN {X 41.474,Y 112.894,Z 53.276,A 180.000,B 0.000,C 180.000} C_DIS
LIN {X 41.593,Y 112.998,Z 53.270,A 180.000,B 0.000,C 180.000} C_DIS
LIN {X 41.651,Y 113.051,Z 53.268,A 180.000,B 0.000,C 180.000} C_DIS
LIN {X 41.762,Y 113.162,Z 53.262,A 180.000,B 0.000,C 180.000} C_DIS
LIN {X 41.929,Y 113.329,Z 53.254,A 180.000,B 0.000,C 180.000} C_DIS
LIN {X 41.984,Y 113.386,Z 53.251,A 180.000,B 0.000,C 180.000} C_DIS
LIN {X 42.140,Y 113.563,Z 53.243,A 180.000,B 0.000,C 180.000} C_DIS
LIN {X 42.244,Y 113.682,Z 53.237,A 180.000,B 0.000,C 180.000} C_DIS
LIN {X 42.295,Y 113.742,Z 53.235,A 180.000,B 0.000,C 180.000} C_DIS
LIN {X 42.391,Y 113.866,Z 53.229,A 180.000,B 0.000,C 180.000} C_DIS
LIN {X 42.536,Y 114.053,Z 53.221,A 180.000,B 0.000,C 180.000} C_DIS
LIN {X 42.583,Y 114.116,Z 53.218,A 180.000,B 0.000,C 180.000} C_DIS
LIN {X 42.716,Y 114.312,Z 53.210,A 180.000,B 0.000,C 180.000} C_DIS
LIN {X 42.804,Y 114.442,Z 53.204,A 180.000,B 0.000,C 180.000} C_DIS
LIN {X 42.847,Y 114.508,Z 53.202,A 180.000,B 0.000,C 180.000} C_DIS
LIN {X 42.927,Y 114.644,Z 53.196,A 180.000,B 0.000,C 180.000} C_DIS
LIN {X 43.007,Y 114.779,Z 53.191,A 180.000,B 0.000,C 180.000} C_DIS
LIN {X 43.047,Y 114.847,Z 53.188,A 180.000,B 0.000,C 180.000} C_DIS
LIN {X 43.086,Y 114.916,Z 53.185,A 180.000,B 0.000,C 180.000} C_DIS
LIN {X 43.157,Y 115.056,Z 53.180,A 180.000,B 0.000,C 180.000} C_DIS
LIN {X 43.229,Y 115.196,Z 53.174,A 180.000,B 0.000,C 180.000} C_DIS
LIN {X 43.264,Y 115.267,Z 53.172,A 180.000,B 0.000,C 180.000} C_DIS
LIN {X 43.298,Y 115.338,Z 53.169,A 180.000,B 0.000,C 180.000} C_DIS
LIN {X 43.361,Y 115.482,Z 53.164,A 180.000,B 0.000,C 180.000} C_DIS
LIN {X 43.392,Y 115.555,Z 53.161,A 180.000,B 0.000,C 180.000} C_DIS
LIN {X 43.423,Y 115.627,Z 53.159,A 180.000,B 0.000,C 180.000} C_DIS
LIN {X 43.455,Y 115.699,Z 53.156,A 180.000,B 0.000,C 180.000} C_DIS
LIN {X 43.484,Y 115.772,Z 53.154,A 180.000,B 0.000,C 180.000} C_DIS
LIN {X 43.511,Y 115.846,Z 53.151,A 180.000,B 0.000,C 180.000} C_DIS
LIN {X 43.537,Y 115.920,Z 53.149,A 180.000,B 0.000,C 180.000} C_DIS
LIN {X 43.591,Y 116.069,Z 53.144,A 180.000,B 0.000,C 180.000} C_DIS
LIN {X 43.642,Y 116.218,Z 53.139,A 180.000,B 0.000,C 180.000} C_DIS
LIN {X 43.686,Y 116.369,Z 53.134,A 180.000,B 0.000,C 180.000} C_DIS
LIN {X 43.730,Y 116.520,Z 53.129,A 180.000,B 0.000,C 180.000} C_DIS
LIN {X 43.771,Y 116.672,Z 53.124,A 180.000,B 0.000,C 180.000} C_DIS
LIN {X 43.806,Y 116.826,Z 53.120,A 180.000,B 0.000,C 180.000} C_DIS
LIN {X 43.840,Y 116.979,Z 53.115,A 180.000,B 0.000,C 180.000} C_DIS
LIN {X 43.872,Y 117.133,Z 53.111,A 180.000,B 0.000,C 180.000} C_DIS
LIN {X 43.897,Y 117.289,Z 53.106,A 180.000,B 0.000,C 180.000} C_DIS
LIN {X 43.921,Y 117.445,Z 53.102,A 180.000,B 0.000,C 180.000} C_DIS
LIN {X 43.943,Y 117.601,Z 53.097,A 180.000,B 0.000,C 180.000} C_DIS
LIN {X 43.958,Y 117.757,Z 53.093,A 180.000,B 0.000,C 180.000} C_DIS
LIN {X 43.973,Y 117.914,Z 53.089,A 180.000,B 0.000,C 180.000} C_DIS
LIN {X 43.985,Y 118.071,Z 53.085,A 180.000,B 0.000,C 180.000} C_DIS
LIN {X 43.990,Y 118.229,Z 53.081,A 180.000,B 0.000,C 180.000} C_DIS
LIN {X 43.995,Y 118.386,Z 53.077,A 180.000,B 0.000,C 180.000} C_DIS
LIN {X 43.997,Y 118.544,Z 53.073,A 180.000,B 0.000,C 180.000} C_DIS
LIN {X 43.992,Y 118.701,Z 53.070,A 180.000,B 0.000,C 180.000} C_DIS
LIN {X 43.988,Y 118.858,Z 53.066,A 180.000,B 0.000,C 180.000} C_DIS
LIN {X 43.980,Y 119.016,Z 53.062,A 180.000,B 0.000,C 180.000} C_DIS
LIN {X 43.965,Y 119.172,Z 53.059,A 180.000,B 0.000,C 180.000} C_DIS
LIN {X 43.950,Y 119.329,Z 53.056,A 180.000,B 0.000,C 180.000} C_DIS
LIN {X 43.932,Y 119.486,Z 53.052,A 180.000,B 0.000,C 180.000} C_DIS
LIN {X 43.908,Y 119.641,Z 53.049,A 180.000,B 0.000,C 180.000} C_DIS
LIN {X 43.883,Y 119.797,Z 53.046,A 180.000,B 0.000,C 180.000} C_DIS
LIN {X 43.855,Y 119.952,Z 53.043,A 180.000,B 0.000,C 180.000} C_DIS
LIN {X 43.821,Y 120.106,Z 53.040,A 180.000,B 0.000,C 180.000} C_DIS
LIN {X 43.787,Y 120.259,Z 53.037,A 180.000,B 0.000,C 180.000} C_DIS
LIN {X 43.749,Y 120.412,Z 53.034,A 180.000,B 0.000,C 180.000} C_DIS
LIN {X 43.705,Y 120.564,Z 53.032,A 180.000,B 0.000,C 180.000} C_DIS
LIN {X 43.662,Y 120.715,Z 53.029,A 180.000,B 0.000,C 180.000} C_DIS
LIN {X 43.615,Y 120.865,Z 53.027,A 180.000,B 0.000,C 180.000} C_DIS
LIN {X 43.508,Y 121.161,Z 53.022,A 180.000,B 0.000,C 180.000} C_DIS
LIN {X 43.389,Y 121.453,Z 53.018,A 180.000,B 0.000,C 180.000} C_DIS
LIN {X 43.261,Y 121.741,Z 53.014,A 180.000,B 0.000,C 180.000} C_DIS
LIN {X 43.118,Y 122.021,Z 53.011,A 180.000,B 0.000,C 180.000} C_DIS
LIN {X 42.963,Y 122.296,Z 53.008,A 180.000,B 0.000,C 180.000} C_DIS
LIN {X 42.800,Y 122.565,Z 53.005,A 180.000,B 0.000,C 180.000} C_DIS
LIN {X 42.622,Y 122.826,Z 53.003,A 180.000,B 0.000,C 180.000} C_DIS
LIN {X 42.434,Y 123.078,Z 53.002,A 180.000,B 0.000,C 180.000} C_DIS
LIN {X 42.238,Y 123.325,Z 53.001,A 180.000,B 0.000,C 180.000} C_DIS
LIN {X 42.030,Y 123.561,Z 53.000,A 180.000,B 0.000,C 180.000} C_DIS
LIN {X 41.870,Y 123.729,Z 53.000,A 180.000,B 0.000,C 180.000} C_DIS
; Cutting Move Starts
LIN {X 41.657,Y 123.943,Z 53.000,A 180.000,B 0.000,C 180.000} C_DIS
LIN {X 41.516,Y 124.070,Z 53.000,A 180.000,B 0.000,C 180.000} C_DIS
LIN {X 41.299,Y 124.261,Z 53.000,A 180.000,B 0.000,C 180.000} C_DIS
LIN {X 41.120,Y 124.402,Z 53.000,A 180.000,B 0.000,C 180.000} C_DIS
LIN {X 40.942,Y 124.540,Z 53.000,A 180.000,B 0.000,C 180.000} C_DIS
LIN {X 40.850,Y 124.606,Z 53.000,A 180.000,B 0.000,C 180.000} C_DIS
LIN {X 40.584,Y 124.787,Z 53.000,A 180.000,B 0.000,C 180.000} C_DIS
LIN {X 40.405,Y 124.898,Z 53.000,A 180.000,B 0.000,C 180.000} C_DIS
LIN {X 40.226,Y 125.004,Z 53.000,A 180.000,B 0.000,C 180.000} C_DIS
LIN {X 40.048,Y 125.104,Z 53.000,A 180.000,B 0.000,C 180.000} C_DIS
LIN {X 39.869,Y 125.195,Z 53.000,A 180.000,B 0.000,C 180.000} C_DIS
LIN {X 39.690,Y 125.286,Z 53.000,A 180.000,B 0.000,C 180.000} C_DIS
LIN {X 39.333,Y 125.441,Z 53.000,A 180.000,B 0.000,C 180.000} C_DIS
LIN {X 39.184,Y 125.500,Z 53.000,A 180.000,B 0.000,C 180.000} C_DIS
LIN {X 38.975,Y 125.575,Z 53.000,A 180.000,B 0.000,C 180.000} C_DIS
LIN {X 38.796,Y 125.638,Z 53.000,A 180.000,B 0.000,C 180.000} C_DIS
LIN {X 38.439,Y 125.742,Z 53.000,A 180.000,B 0.000,C 180.000} C_DIS
LIN {X 38.260,Y 125.787,Z 53.000,A 180.000,B 0.000,C 180.000} C_DIS
LIN {X 37.944,Y 125.857,Z 53.000,A 180.000,B 0.000,C 180.000} C_DIS
LIN {X 37.902,Y 125.866,Z 53.000,A 180.000,B 0.000,C 180.000} C_DIS
LIN {X 37.545,Y 125.923,Z 53.000,A 180.000,B 0.000,C 180.000} C_DIS
LIN {X 37.366,Y 125.947,Z 53.000,A 180.000,B 0.000,C 180.000} C_DIS
LIN {X 37.009,Y 125.980,Z 53.000,A 180.000,B 0.000,C 180.000} C_DIS
LIN {X 36.830,Y 125.988,Z 53.000,A 180.000,B 0.000,C 180.000} C_DIS
LIN {X 36.651,Y 125.994,Z 53.000,A 180.000,B 0.000,C 180.000} C_DIS
LIN {X 36.472,Y 125.998,Z 53.000,A 180.000,B 0.000,C 180.000} C_DIS
LIN {X 36.115,Y 125.987,Z 53.000,A 180.000,B 0.000,C 180.000} C_DIS
LIN {X 35.936,Y 125.975,Z 53.000,A 180.000,B 0.000,C 180.000} C_DIS
LIN {X 35.578,Y 125.941,Z 53.000,A 180.000,B 0.000,C 180.000} C_DIS
